// TwinCAT 3 PLC project PLC_LMP_VAC_current
// Title: LAMP PLC
// Author: A. Wallace, J. Yin and S. Stubbs
// Description: This version includes a longer needle valve purge time. Updated purge logic to quit the purge incase the interlocks on either VCN 40 VGP 40 or VIC 80 fail.
// ProgramVersion: 3.1.4020.1
// libraries:
//   LCLSVacuumLib,newest,SLAC
//   LCLSVacuumSerialDriverLib,newest,SLAC
//   Tc2_Standard,3.3.1.0,Beckhoff Automation GmbH
//   Tc2_SUPS,newest,Beckhoff Automation GmbH
//   Tc2_System,3.3.10.0,Beckhoff Automation GmbH
//   Tc2_Utilities,3.3.11.0,Beckhoff Automation GmbH
//   Tc3_Interfaces,3.3.0.0,Beckhoff Automation GmbH
//   Standard, * (System)
//   Tc2_SerialCom, * (Beckhoff Automation GmbH)
//   Tc3_Module, * (Beckhoff Automation GmbH)
// project tree:
//   Global Variables/ GVL.TcGVL, GVL_Autosave.TcGVL, GVL_COM_Buffers.TcGVL, GVL_Devices.TcGVL, GVL_IO.TcGVL, GVL_SerialIO.TcGVL
//   POUs/ Ext_Interlocks.TcPOU, MAIN.TcPOU, p_Initialize.TcPOU, p_SoftIOMap.TcPOU, p_ModbusMapRx.TcPOU, p_ModbusMapTx.TcPOU, p_GaugeSup.TcPOU, p_PTMSup.TcPOU, p_ValveSup.TcPOU, Encoders.TcPOU, p_Autosave.TcPOU, P_Serial_Com.TcPOU, P_Serial_PTM_IO.TcPOU
//   POUs/Functions/ FB_VRC_LAMP.TcPOU
//   / Standard.TcTTO, SerialIO.TcTTO
// real-time tasks:
//   TASK Standard: cycle T#10ms, priority 8, ADS port 351
//   TASK SerialIO: cycle T#5ms, priority 6, ADS port 352
// I/O:
//   DEVICE LAMP Fieldbus (EtherCAT), AmsNetId 5.21.50.18.2.1
//     Term 1 (EK1200) [EK1200-5000 EtherCAT Power supply (2A E-Bus)]
//       Term 2 (EL3064) [EL3064 4Ch. Ana. Input 0-10V]
//       Term 3 (EL3064) [EL3064 4Ch. Ana. Input 0-10V]
//       Term 4 (EL1008) [EL1008 8Ch. Dig. Input 24V, 3ms]
//       Term 5 (EL2008) [EL2008 8Ch. Dig. Output 24V, 0.5A]
//       Term 6 (EL2798) [EL2798 8Ch. Dig. Output 24V AC/DC, 2A, potential-free]
//       Term 7 (EL6731) [EL6731 PROFIBUS DP Master] (disabled)
//       Term 8 (EK1110) [EK1110 EtherCAT extension]
//     R10_A (EP6002-0002) [EP6002-0002 Interface (RS232/422/485)]
//     R10_B (EP6002-0002) [EP6002-0002 Interface (RS232/422/485)]
//     IC1-EB1 (EP6002-0002) [EP6002-0002 Interface (RS232/422/485)]
//     IC1-EB2 (EP3174-0002) [EP3174-0002 4Ch. Ana. Input +/-10V, 0-10V, 0/4-20mA configurable]
//     IC1-EB3 (EP2624-0002) [EP2624-0002 4Ch. Relay Output, NO (125V AC / 30V DC)]
//     IC1-EB4 (EP2339-0021) [EP2339-0021 16 Ch. Dig. Input/Output 24V, 0,5A, M8]
//     DET-EB1 (EP6002-0002) [EP6002-0002 Interface (RS232/422/485)]
//     DET-EB2 (EP3174-0002) [EP3174-0002 4Ch. Ana. Input +/-10V, 0-10V, 0/4-20mA configurable]
//     DET-EB3 (EP2624-0002) [EP2624-0002 4Ch. Relay Output, NO (125V AC / 30V DC)]
//     DET-EB4 (EP2339-0021) [EP2339-0021 16 Ch. Dig. Input/Output 24V, 0,5A, M8]
//     DET-EB5 (EP2624-0002) [EP2624-0002 4Ch. Relay Output, NO (125V AC / 30V DC)]
//     GJ1-EB1 (EP2624-0002) [EP2624-0002 4Ch. Relay Output, NO (125V AC / 30V DC)]
//     GJ-EB2 (EP3174-0002) [EP3174-0002 4Ch. Ana. Input +/-10V, 0-10V, 0/4-20mA configurable]
//     GJ-EB3 (EP2339-0021) [EP2339-0021 16 Ch. Dig. Input/Output 24V, 0,5A, M8]
//     GJ-EB4 (EP3174-0002) [EP3174-0002 4Ch. Ana. Input +/-10V, 0-10V, 0/4-20mA, +/-10mA configurable]
//     LRS-EB1 (EP3174-0002) [EP3174-0002 4Ch. Ana. Input +/-10V, 0-10V, 0/4-20mA configurable]
//     LRS-EB2 (EP3174-0002) [EP3174-0002 4Ch. Ana. Input +/-10V, 0-10V, 0/4-20mA, +/-10mA configurable]
//     LRS-EB3 (EP2339-0021) [EP2339-0021 16 Ch. Dig. Input/Output 24V, 0,5A, M8]
//     LRS-EB4 (EP2339-0021) [EP2339-0021 16 Ch. Dig. Input/Output 24V, 0,5A, M8]
//     H2E-EB1 (EP2339-0021) [EP2339-0021 16 Ch. Dig. Input/Output 24V, 0,5A, M8] (disabled)
//     H2E-EB2 (EP3174-0002) [EP3174-0002 4Ch. Ana. Input +/-10V, 0-10V, 0/4-20mA, +/-10mA configurable] (disabled)
//   DEVICE LAMP(EtherCAT Slave), AmsNetId 5.21.50.18.4.255
//   DEVICE Device 2 (EL6731) (disabled), AmsNetId 5.21.50.18.3.1
// variable links:
//   PLC_LMP_VAC_current/PLC_LMP_VAC_current Instance <-> LAMP Fieldbus (EtherCAT)/DET-EB1 (EP6002-0002)
//     SerialIO Inputs/GVL_SerialIO.DET_P1_stComIn/D[0] <-> COM TxPDO-Map Inputs Channel 1/Data In 0
//     SerialIO Inputs/GVL_SerialIO.DET_P1_stComIn/D[10] <-> COM TxPDO-Map Inputs Channel 1/Data In 10
//     SerialIO Inputs/GVL_SerialIO.DET_P1_stComIn/D[11] <-> COM TxPDO-Map Inputs Channel 1/Data In 11
//     SerialIO Inputs/GVL_SerialIO.DET_P1_stComIn/D[12] <-> COM TxPDO-Map Inputs Channel 1/Data In 12
//     SerialIO Inputs/GVL_SerialIO.DET_P1_stComIn/D[13] <-> COM TxPDO-Map Inputs Channel 1/Data In 13
//     SerialIO Inputs/GVL_SerialIO.DET_P1_stComIn/D[14] <-> COM TxPDO-Map Inputs Channel 1/Data In 14
//     SerialIO Inputs/GVL_SerialIO.DET_P1_stComIn/D[15] <-> COM TxPDO-Map Inputs Channel 1/Data In 15
//     SerialIO Inputs/GVL_SerialIO.DET_P1_stComIn/D[16] <-> COM TxPDO-Map Inputs Channel 1/Data In 16
//     SerialIO Inputs/GVL_SerialIO.DET_P1_stComIn/D[17] <-> COM TxPDO-Map Inputs Channel 1/Data In 17
//     SerialIO Inputs/GVL_SerialIO.DET_P1_stComIn/D[18] <-> COM TxPDO-Map Inputs Channel 1/Data In 18
//     SerialIO Inputs/GVL_SerialIO.DET_P1_stComIn/D[19] <-> COM TxPDO-Map Inputs Channel 1/Data In 19
//     SerialIO Inputs/GVL_SerialIO.DET_P1_stComIn/D[1] <-> COM TxPDO-Map Inputs Channel 1/Data In 1
//     SerialIO Inputs/GVL_SerialIO.DET_P1_stComIn/D[20] <-> COM TxPDO-Map Inputs Channel 1/Data In 20
//     SerialIO Inputs/GVL_SerialIO.DET_P1_stComIn/D[21] <-> COM TxPDO-Map Inputs Channel 1/Data In 21
//     SerialIO Inputs/GVL_SerialIO.DET_P1_stComIn/D[2] <-> COM TxPDO-Map Inputs Channel 1/Data In 2
//     SerialIO Inputs/GVL_SerialIO.DET_P1_stComIn/D[3] <-> COM TxPDO-Map Inputs Channel 1/Data In 3
//     SerialIO Inputs/GVL_SerialIO.DET_P1_stComIn/D[4] <-> COM TxPDO-Map Inputs Channel 1/Data In 4
//     SerialIO Inputs/GVL_SerialIO.DET_P1_stComIn/D[5] <-> COM TxPDO-Map Inputs Channel 1/Data In 5
//     SerialIO Inputs/GVL_SerialIO.DET_P1_stComIn/D[6] <-> COM TxPDO-Map Inputs Channel 1/Data In 6
//     SerialIO Inputs/GVL_SerialIO.DET_P1_stComIn/D[7] <-> COM TxPDO-Map Inputs Channel 1/Data In 7
//     SerialIO Inputs/GVL_SerialIO.DET_P1_stComIn/D[8] <-> COM TxPDO-Map Inputs Channel 1/Data In 8
//     SerialIO Inputs/GVL_SerialIO.DET_P1_stComIn/D[9] <-> COM TxPDO-Map Inputs Channel 1/Data In 9
//     SerialIO Inputs/GVL_SerialIO.DET_P2_stComIn/D[0] <-> COM TxPDO-Map Inputs Channel 2/Data In 0
//     SerialIO Inputs/GVL_SerialIO.DET_P2_stComIn/D[10] <-> COM TxPDO-Map Inputs Channel 2/Data In 10
//     SerialIO Inputs/GVL_SerialIO.DET_P2_stComIn/D[11] <-> COM TxPDO-Map Inputs Channel 2/Data In 11
//     SerialIO Inputs/GVL_SerialIO.DET_P2_stComIn/D[12] <-> COM TxPDO-Map Inputs Channel 2/Data In 12
//     SerialIO Inputs/GVL_SerialIO.DET_P2_stComIn/D[13] <-> COM TxPDO-Map Inputs Channel 2/Data In 13
//     SerialIO Inputs/GVL_SerialIO.DET_P2_stComIn/D[14] <-> COM TxPDO-Map Inputs Channel 2/Data In 14
//     SerialIO Inputs/GVL_SerialIO.DET_P2_stComIn/D[15] <-> COM TxPDO-Map Inputs Channel 2/Data In 15
//     SerialIO Inputs/GVL_SerialIO.DET_P2_stComIn/D[16] <-> COM TxPDO-Map Inputs Channel 2/Data In 16
//     SerialIO Inputs/GVL_SerialIO.DET_P2_stComIn/D[17] <-> COM TxPDO-Map Inputs Channel 2/Data In 17
//     SerialIO Inputs/GVL_SerialIO.DET_P2_stComIn/D[18] <-> COM TxPDO-Map Inputs Channel 2/Data In 18
//     SerialIO Inputs/GVL_SerialIO.DET_P2_stComIn/D[19] <-> COM TxPDO-Map Inputs Channel 2/Data In 19
//     SerialIO Inputs/GVL_SerialIO.DET_P2_stComIn/D[1] <-> COM TxPDO-Map Inputs Channel 2/Data In 1
//     SerialIO Inputs/GVL_SerialIO.DET_P2_stComIn/D[20] <-> COM TxPDO-Map Inputs Channel 2/Data In 20
//     SerialIO Inputs/GVL_SerialIO.DET_P2_stComIn/D[21] <-> COM TxPDO-Map Inputs Channel 2/Data In 21
//     SerialIO Inputs/GVL_SerialIO.DET_P2_stComIn/D[2] <-> COM TxPDO-Map Inputs Channel 2/Data In 2
//     SerialIO Inputs/GVL_SerialIO.DET_P2_stComIn/D[3] <-> COM TxPDO-Map Inputs Channel 2/Data In 3
//     SerialIO Inputs/GVL_SerialIO.DET_P2_stComIn/D[4] <-> COM TxPDO-Map Inputs Channel 2/Data In 4
//     SerialIO Inputs/GVL_SerialIO.DET_P2_stComIn/D[5] <-> COM TxPDO-Map Inputs Channel 2/Data In 5
//     SerialIO Inputs/GVL_SerialIO.DET_P2_stComIn/D[6] <-> COM TxPDO-Map Inputs Channel 2/Data In 6
//     SerialIO Inputs/GVL_SerialIO.DET_P2_stComIn/D[7] <-> COM TxPDO-Map Inputs Channel 2/Data In 7
//     SerialIO Inputs/GVL_SerialIO.DET_P2_stComIn/D[8] <-> COM TxPDO-Map Inputs Channel 2/Data In 8
//     SerialIO Inputs/GVL_SerialIO.DET_P2_stComIn/D[9] <-> COM TxPDO-Map Inputs Channel 2/Data In 9
//     SerialIO Inputs/GVL_SerialIO.DET_P1_stComIn/Status <-> COM TxPDO-Map Inputs Channel 1/Status
//     SerialIO Inputs/GVL_SerialIO.DET_P2_stComIn/Status <-> COM TxPDO-Map Inputs Channel 2/Status
//     SerialIO Outputs/GVL_SerialIO.DET_P1_stComOut/Ctrl <-> COM RxPDO-Map Outputs Channel 1/Ctrl
//     SerialIO Outputs/GVL_SerialIO.DET_P2_stComOut/Ctrl <-> COM RxPDO-Map Outputs Channel 2/Ctrl
//     SerialIO Outputs/GVL_SerialIO.DET_P1_stComOut/D[0] <-> COM RxPDO-Map Outputs Channel 1/Data Out 0
//     SerialIO Outputs/GVL_SerialIO.DET_P1_stComOut/D[10] <-> COM RxPDO-Map Outputs Channel 1/Data Out 10
//     SerialIO Outputs/GVL_SerialIO.DET_P1_stComOut/D[11] <-> COM RxPDO-Map Outputs Channel 1/Data Out 11
//     SerialIO Outputs/GVL_SerialIO.DET_P1_stComOut/D[12] <-> COM RxPDO-Map Outputs Channel 1/Data Out 12
//     SerialIO Outputs/GVL_SerialIO.DET_P1_stComOut/D[13] <-> COM RxPDO-Map Outputs Channel 1/Data Out 13
//     SerialIO Outputs/GVL_SerialIO.DET_P1_stComOut/D[14] <-> COM RxPDO-Map Outputs Channel 1/Data Out 14
//     SerialIO Outputs/GVL_SerialIO.DET_P1_stComOut/D[15] <-> COM RxPDO-Map Outputs Channel 1/Data Out 15
//     SerialIO Outputs/GVL_SerialIO.DET_P1_stComOut/D[16] <-> COM RxPDO-Map Outputs Channel 1/Data Out 16
//     SerialIO Outputs/GVL_SerialIO.DET_P1_stComOut/D[17] <-> COM RxPDO-Map Outputs Channel 1/Data Out 17
//     SerialIO Outputs/GVL_SerialIO.DET_P1_stComOut/D[18] <-> COM RxPDO-Map Outputs Channel 1/Data Out 18
//     SerialIO Outputs/GVL_SerialIO.DET_P1_stComOut/D[19] <-> COM RxPDO-Map Outputs Channel 1/Data Out 19
//     SerialIO Outputs/GVL_SerialIO.DET_P1_stComOut/D[1] <-> COM RxPDO-Map Outputs Channel 1/Data Out 1
//     SerialIO Outputs/GVL_SerialIO.DET_P1_stComOut/D[20] <-> COM RxPDO-Map Outputs Channel 1/Data Out 20
//     SerialIO Outputs/GVL_SerialIO.DET_P1_stComOut/D[21] <-> COM RxPDO-Map Outputs Channel 1/Data Out 21
//     SerialIO Outputs/GVL_SerialIO.DET_P1_stComOut/D[2] <-> COM RxPDO-Map Outputs Channel 1/Data Out 2
//     SerialIO Outputs/GVL_SerialIO.DET_P1_stComOut/D[3] <-> COM RxPDO-Map Outputs Channel 1/Data Out 3
//     SerialIO Outputs/GVL_SerialIO.DET_P1_stComOut/D[4] <-> COM RxPDO-Map Outputs Channel 1/Data Out 4
//     SerialIO Outputs/GVL_SerialIO.DET_P1_stComOut/D[5] <-> COM RxPDO-Map Outputs Channel 1/Data Out 5
//     SerialIO Outputs/GVL_SerialIO.DET_P1_stComOut/D[6] <-> COM RxPDO-Map Outputs Channel 1/Data Out 6
//     SerialIO Outputs/GVL_SerialIO.DET_P1_stComOut/D[7] <-> COM RxPDO-Map Outputs Channel 1/Data Out 7
//     SerialIO Outputs/GVL_SerialIO.DET_P1_stComOut/D[8] <-> COM RxPDO-Map Outputs Channel 1/Data Out 8
//     SerialIO Outputs/GVL_SerialIO.DET_P1_stComOut/D[9] <-> COM RxPDO-Map Outputs Channel 1/Data Out 9
//     SerialIO Outputs/GVL_SerialIO.DET_P2_stComOut/D[0] <-> COM RxPDO-Map Outputs Channel 2/Data Out 0
//     SerialIO Outputs/GVL_SerialIO.DET_P2_stComOut/D[10] <-> COM RxPDO-Map Outputs Channel 2/Data Out 10
//     SerialIO Outputs/GVL_SerialIO.DET_P2_stComOut/D[11] <-> COM RxPDO-Map Outputs Channel 2/Data Out 11
//     SerialIO Outputs/GVL_SerialIO.DET_P2_stComOut/D[12] <-> COM RxPDO-Map Outputs Channel 2/Data Out 12
//     SerialIO Outputs/GVL_SerialIO.DET_P2_stComOut/D[13] <-> COM RxPDO-Map Outputs Channel 2/Data Out 13
//     SerialIO Outputs/GVL_SerialIO.DET_P2_stComOut/D[14] <-> COM RxPDO-Map Outputs Channel 2/Data Out 14
//     SerialIO Outputs/GVL_SerialIO.DET_P2_stComOut/D[15] <-> COM RxPDO-Map Outputs Channel 2/Data Out 15
//     SerialIO Outputs/GVL_SerialIO.DET_P2_stComOut/D[16] <-> COM RxPDO-Map Outputs Channel 2/Data Out 16
//     SerialIO Outputs/GVL_SerialIO.DET_P2_stComOut/D[17] <-> COM RxPDO-Map Outputs Channel 2/Data Out 17
//     SerialIO Outputs/GVL_SerialIO.DET_P2_stComOut/D[18] <-> COM RxPDO-Map Outputs Channel 2/Data Out 18
//     SerialIO Outputs/GVL_SerialIO.DET_P2_stComOut/D[19] <-> COM RxPDO-Map Outputs Channel 2/Data Out 19
//     SerialIO Outputs/GVL_SerialIO.DET_P2_stComOut/D[1] <-> COM RxPDO-Map Outputs Channel 2/Data Out 1
//     SerialIO Outputs/GVL_SerialIO.DET_P2_stComOut/D[20] <-> COM RxPDO-Map Outputs Channel 2/Data Out 20
//     SerialIO Outputs/GVL_SerialIO.DET_P2_stComOut/D[21] <-> COM RxPDO-Map Outputs Channel 2/Data Out 21
//     SerialIO Outputs/GVL_SerialIO.DET_P2_stComOut/D[2] <-> COM RxPDO-Map Outputs Channel 2/Data Out 2
//     SerialIO Outputs/GVL_SerialIO.DET_P2_stComOut/D[3] <-> COM RxPDO-Map Outputs Channel 2/Data Out 3
//     SerialIO Outputs/GVL_SerialIO.DET_P2_stComOut/D[4] <-> COM RxPDO-Map Outputs Channel 2/Data Out 4
//     SerialIO Outputs/GVL_SerialIO.DET_P2_stComOut/D[5] <-> COM RxPDO-Map Outputs Channel 2/Data Out 5
//     SerialIO Outputs/GVL_SerialIO.DET_P2_stComOut/D[6] <-> COM RxPDO-Map Outputs Channel 2/Data Out 6
//     SerialIO Outputs/GVL_SerialIO.DET_P2_stComOut/D[7] <-> COM RxPDO-Map Outputs Channel 2/Data Out 7
//     SerialIO Outputs/GVL_SerialIO.DET_P2_stComOut/D[8] <-> COM RxPDO-Map Outputs Channel 2/Data Out 8
//     SerialIO Outputs/GVL_SerialIO.DET_P2_stComOut/D[9] <-> COM RxPDO-Map Outputs Channel 2/Data Out 9
//   PLC_LMP_VAC_current/PLC_LMP_VAC_current Instance <-> LAMP Fieldbus (EtherCAT)/DET-EB2 (EP3174-0002)
//     Standard Inputs/GVL_IO.AI_DET_EB2Ch01 <-> AI Standard Channel 1/Value
//     Standard Inputs/GVL_IO.AI_DET_EB2Ch02 <-> AI Standard Channel 2/Value
//     Standard Inputs/GVL_IO.AI_DET_EB2Ch03 <-> AI Standard Channel 3/Value
//     Standard Inputs/GVL_IO.AI_DET_EB2Ch04 <-> AI Standard Channel 4/Value
//   PLC_LMP_VAC_current/PLC_LMP_VAC_current Instance <-> LAMP Fieldbus (EtherCAT)/DET-EB3 (EP2624-0002)
//     Standard Outputs/GVL_IO.RelayO_DET_EB3Ch01 <-> Channel 1/Output
//     Standard Outputs/GVL_IO.RelayO_DET_EB3Ch02 <-> Channel 2/Output
//     Standard Outputs/GVL_IO.RelayO_DET_EB3Ch03 <-> Channel 3/Output
//     Standard Outputs/GVL_IO.RelayO_DET_EB3Ch04 <-> Channel 4/Output
//   PLC_LMP_VAC_current/PLC_LMP_VAC_current Instance <-> LAMP Fieldbus (EtherCAT)/DET-EB4 (EP2339-0021)
//     Standard Inputs/GVL_IO.DiscIO_DET_EB4Ch02 <-> Channel 2/Input
//     Standard Inputs/GVL_IO.DiscIO_DET_EB4Ch03 <-> Channel 3/Input
//     Standard Inputs/GVL_IO.DiscIO_DET_EB4Ch05 <-> Channel 5/Input
//     Standard Inputs/GVL_IO.DiscIO_DET_EB4Ch06 <-> Channel 6/Input
//     Standard Inputs/GVL_IO.DiscIO_DET_EB4Ch08 <-> Channel 8/Input
//     Standard Inputs/GVL_IO.DiscIO_DET_EB4Ch09 <-> Channel 9/Input
//     Standard Inputs/GVL_IO.DiscIO_DET_EB4Ch11 <-> Channel 11/Input
//     Standard Inputs/GVL_IO.DiscIO_DET_EB4Ch12 <-> Channel 12/Input
//     Standard Inputs/GVL_IO.DiscIO_DET_EB4Ch14 <-> Channel 14/Input
//     Standard Inputs/GVL_IO.DiscIO_DET_EB4Ch15 <-> Channel 15/Input
//     Standard Inputs/GVL_IO.DiscIO_DET_EB4Ch16 <-> Channel 16/Input
//     Standard Outputs/GVL_IO.DiscIO_DET_EB4Ch01 <-> Channel 17/Output
//     Standard Outputs/GVL_IO.DiscIO_DET_EB4Ch04 <-> Channel 20/Output
//     Standard Outputs/GVL_IO.DiscIO_DET_EB4Ch07 <-> Channel 23/Output
//     Standard Outputs/GVL_IO.DiscIO_DET_EB4Ch10 <-> Channel 26/Output
//     Standard Outputs/GVL_IO.DiscIO_DET_EB4Ch13 <-> Channel 29/Output
//   PLC_LMP_VAC_current/PLC_LMP_VAC_current Instance <-> LAMP Fieldbus (EtherCAT)/DET-EB5 (EP2624-0002)
//     Standard Outputs/GVL_IO.RelayO_DET_EB5Ch01 <-> Channel 1/Output
//     Standard Outputs/GVL_IO.RelayO_DET_EB5Ch02 <-> Channel 2/Output
//     Standard Outputs/GVL_IO.RelayO_DET_EB5Ch03 <-> Channel 3/Output
//     Standard Outputs/GVL_IO.RelayO_DET_EB5Ch04 <-> Channel 4/Output
//   PLC_LMP_VAC_current/PLC_LMP_VAC_current Instance <-> LAMP Fieldbus (EtherCAT)/GJ-EB2 (EP3174-0002)
//     Standard Inputs/GVL_IO.AI_GJ_EB2Ch01 <-> AI Standard Channel 1/Value
//     Standard Inputs/GVL_IO.AI_GJ_EB2Ch02 <-> AI Standard Channel 2/Value
//     Standard Inputs/GVL_IO.AI_GJ_EB2Ch03 <-> AI Standard Channel 3/Value
//     Standard Inputs/GVL_IO.AI_GJ_EB2Ch04 <-> AI Standard Channel 4/Value
//   PLC_LMP_VAC_current/PLC_LMP_VAC_current Instance <-> LAMP Fieldbus (EtherCAT)/GJ-EB3 (EP2339-0021)
//     Standard Inputs/GVL_IO.DiscIO_GJ_EB3Ch02 <-> Channel 2/Input
//     Standard Inputs/GVL_IO.DiscIO_GJ_EB3Ch03 <-> Channel 3/Input
//     Standard Inputs/GVL_IO.DiscIO_GJ_EB3Ch05 <-> Channel 5/Input
//     Standard Inputs/GVL_IO.DiscIO_GJ_EB3Ch06 <-> Channel 6/Input
//     Standard Inputs/GVL_IO.DiscIO_GJ_EB3Ch08 <-> Channel 8/Input
//     Standard Inputs/GVL_IO.DiscIO_GJ_EB3Ch09 <-> Channel 9/Input
//     Standard Inputs/GVL_IO.DiscIO_GJ_EB3Ch11 <-> Channel 11/Input
//     Standard Inputs/GVL_IO.DiscIO_GJ_EB3Ch12 <-> Channel 12/Input
//     Standard Inputs/GVL_IO.DiscIO_GJ_EB3Ch14 <-> Channel 14/Input
//     Standard Inputs/GVL_IO.DiscIO_GJ_EB3Ch15 <-> Channel 15/Input
//     Standard Inputs/GVL_IO.DiscIO_GJ_EB3Ch16 <-> Channel 16/Input
//     Standard Outputs/GVL_IO.DiscIO_GJ_EB3Ch01 <-> Channel 17/Output
//     Standard Outputs/GVL_IO.DiscIO_GJ_EB3Ch04 <-> Channel 20/Output
//     Standard Outputs/GVL_IO.DiscIO_GJ_EB3Ch07 <-> Channel 23/Output
//     Standard Outputs/GVL_IO.DiscIO_GJ_EB3Ch10 <-> Channel 26/Output
//     Standard Outputs/GVL_IO.DiscIO_GJ_EB3Ch13 <-> Channel 29/Output
//   PLC_LMP_VAC_current/PLC_LMP_VAC_current Instance <-> LAMP Fieldbus (EtherCAT)/GJ-EB4 (EP3174-0002)
//     Standard Inputs/GVL_IO.AI_GJ_EB4Ch01 <-> AI Standard Channel 1/Value
//     Standard Inputs/GVL_IO.AI_GJ_EB4Ch02 <-> AI Standard Channel 2/Value
//     Standard Inputs/GVL_IO.AI_GJ_EB4Ch03 <-> AI Standard Channel 3/Value
//     Standard Inputs/GVL_IO.AI_GJ_EB4Ch04 <-> AI Standard Channel 4/Value
//   PLC_LMP_VAC_current/PLC_LMP_VAC_current Instance <-> LAMP Fieldbus (EtherCAT)/GJ1-EB1 (EP2624-0002)
//     Standard Outputs/GVL_IO.RelayO_GJ_EB1Ch01 <-> Channel 1/Output
//     Standard Outputs/GVL_IO.RelayO_GJ_EB1Ch02 <-> Channel 2/Output
//     Standard Outputs/GVL_IO.RelayO_GJ_EB1Ch03 <-> Channel 3/Output
//     Standard Outputs/GVL_IO.RelayO_GJ_EB1Ch04 <-> Channel 4/Output
//   PLC_LMP_VAC_current/PLC_LMP_VAC_current Instance <-> LAMP Fieldbus (EtherCAT)/H2E-EB1 (EP2339-0021)
//     Standard Inputs/GVL_IO.DiscIO_H2E_EB1Ch02 <-> Channel 2/Input
//     Standard Inputs/GVL_IO.DiscIO_H2E_EB1Ch03 <-> Channel 3/Input
//     Standard Inputs/GVL_IO.DiscIO_H2E_EB1Ch05 <-> Channel 5/Input
//     Standard Inputs/GVL_IO.DiscIO_H2E_EB1Ch06 <-> Channel 6/Input
//     Standard Inputs/GVL_IO.DiscIO_H2E_EB1Ch08 <-> Channel 8/Input
//     Standard Inputs/GVL_IO.DiscIO_H2E_EB1Ch09 <-> Channel 9/Input
//     Standard Inputs/GVL_IO.DiscIO_H2E_EB1Ch11 <-> Channel 11/Input
//     Standard Inputs/GVL_IO.DiscIO_H2E_EB1Ch12 <-> Channel 12/Input
//     Standard Inputs/GVL_IO.DiscIO_H2E_EB1Ch14 <-> Channel 14/Input
//     Standard Inputs/GVL_IO.DiscIO_H2E_EB1Ch15 <-> Channel 15/Input
//     Standard Inputs/GVL_IO.DiscIO_H2E_EB1Ch16 <-> Channel 16/Input
//     Standard Outputs/GVL_IO.DiscIO_H2E_EB1Ch01 <-> Channel 17/Output
//     Standard Outputs/GVL_IO.DiscIO_H2E_EB1Ch04 <-> Channel 20/Output
//     Standard Outputs/GVL_IO.DiscIO_H2E_EB1Ch07 <-> Channel 23/Output
//     Standard Outputs/GVL_IO.DiscIO_H2E_EB1Ch10 <-> Channel 26/Output
//     Standard Outputs/GVL_IO.DiscIO_H2E_EB1Ch13 <-> Channel 29/Output
//   PLC_LMP_VAC_current/PLC_LMP_VAC_current Instance <-> LAMP Fieldbus (EtherCAT)/H2E-EB2 (EP3174-0002)
//     Standard Inputs/GVL_IO.AI_H2E_EB2Ch01 <-> AI Standard Channel 1/Value
//     Standard Inputs/GVL_IO.AI_H2E_EB2Ch02 <-> AI Standard Channel 2/Value
//     Standard Inputs/GVL_IO.AI_H2E_EB2Ch03 <-> AI Standard Channel 3/Value
//     Standard Inputs/GVL_IO.AI_H2E_EB2Ch04 <-> AI Standard Channel 4/Value
//   PLC_LMP_VAC_current/PLC_LMP_VAC_current Instance <-> LAMP Fieldbus (EtherCAT)/IC1-EB1 (EP6002-0002)
//     SerialIO Inputs/GVL_SerialIO.IC_P1_stComIn/D[0] <-> COM TxPDO-Map Inputs Channel 1/Data In 0
//     SerialIO Inputs/GVL_SerialIO.IC_P1_stComIn/D[10] <-> COM TxPDO-Map Inputs Channel 1/Data In 10
//     SerialIO Inputs/GVL_SerialIO.IC_P1_stComIn/D[11] <-> COM TxPDO-Map Inputs Channel 1/Data In 11
//     SerialIO Inputs/GVL_SerialIO.IC_P1_stComIn/D[12] <-> COM TxPDO-Map Inputs Channel 1/Data In 12
//     SerialIO Inputs/GVL_SerialIO.IC_P1_stComIn/D[13] <-> COM TxPDO-Map Inputs Channel 1/Data In 13
//     SerialIO Inputs/GVL_SerialIO.IC_P1_stComIn/D[14] <-> COM TxPDO-Map Inputs Channel 1/Data In 14
//     SerialIO Inputs/GVL_SerialIO.IC_P1_stComIn/D[15] <-> COM TxPDO-Map Inputs Channel 1/Data In 15
//     SerialIO Inputs/GVL_SerialIO.IC_P1_stComIn/D[16] <-> COM TxPDO-Map Inputs Channel 1/Data In 16
//     SerialIO Inputs/GVL_SerialIO.IC_P1_stComIn/D[17] <-> COM TxPDO-Map Inputs Channel 1/Data In 17
//     SerialIO Inputs/GVL_SerialIO.IC_P1_stComIn/D[18] <-> COM TxPDO-Map Inputs Channel 1/Data In 18
//     SerialIO Inputs/GVL_SerialIO.IC_P1_stComIn/D[19] <-> COM TxPDO-Map Inputs Channel 1/Data In 19
//     SerialIO Inputs/GVL_SerialIO.IC_P1_stComIn/D[1] <-> COM TxPDO-Map Inputs Channel 1/Data In 1
//     SerialIO Inputs/GVL_SerialIO.IC_P1_stComIn/D[20] <-> COM TxPDO-Map Inputs Channel 1/Data In 20
//     SerialIO Inputs/GVL_SerialIO.IC_P1_stComIn/D[21] <-> COM TxPDO-Map Inputs Channel 1/Data In 21
//     SerialIO Inputs/GVL_SerialIO.IC_P1_stComIn/D[2] <-> COM TxPDO-Map Inputs Channel 1/Data In 2
//     SerialIO Inputs/GVL_SerialIO.IC_P1_stComIn/D[3] <-> COM TxPDO-Map Inputs Channel 1/Data In 3
//     SerialIO Inputs/GVL_SerialIO.IC_P1_stComIn/D[4] <-> COM TxPDO-Map Inputs Channel 1/Data In 4
//     SerialIO Inputs/GVL_SerialIO.IC_P1_stComIn/D[5] <-> COM TxPDO-Map Inputs Channel 1/Data In 5
//     SerialIO Inputs/GVL_SerialIO.IC_P1_stComIn/D[6] <-> COM TxPDO-Map Inputs Channel 1/Data In 6
//     SerialIO Inputs/GVL_SerialIO.IC_P1_stComIn/D[7] <-> COM TxPDO-Map Inputs Channel 1/Data In 7
//     SerialIO Inputs/GVL_SerialIO.IC_P1_stComIn/D[8] <-> COM TxPDO-Map Inputs Channel 1/Data In 8
//     SerialIO Inputs/GVL_SerialIO.IC_P1_stComIn/D[9] <-> COM TxPDO-Map Inputs Channel 1/Data In 9
//     SerialIO Inputs/GVL_SerialIO.IC_P2_stComIn/D[0] <-> COM TxPDO-Map Inputs Channel 2/Data In 0
//     SerialIO Inputs/GVL_SerialIO.IC_P2_stComIn/D[10] <-> COM TxPDO-Map Inputs Channel 2/Data In 10
//     SerialIO Inputs/GVL_SerialIO.IC_P2_stComIn/D[11] <-> COM TxPDO-Map Inputs Channel 2/Data In 11
//     SerialIO Inputs/GVL_SerialIO.IC_P2_stComIn/D[12] <-> COM TxPDO-Map Inputs Channel 2/Data In 12
//     SerialIO Inputs/GVL_SerialIO.IC_P2_stComIn/D[13] <-> COM TxPDO-Map Inputs Channel 2/Data In 13
//     SerialIO Inputs/GVL_SerialIO.IC_P2_stComIn/D[14] <-> COM TxPDO-Map Inputs Channel 2/Data In 14
//     SerialIO Inputs/GVL_SerialIO.IC_P2_stComIn/D[15] <-> COM TxPDO-Map Inputs Channel 2/Data In 15
//     SerialIO Inputs/GVL_SerialIO.IC_P2_stComIn/D[16] <-> COM TxPDO-Map Inputs Channel 2/Data In 16
//     SerialIO Inputs/GVL_SerialIO.IC_P2_stComIn/D[17] <-> COM TxPDO-Map Inputs Channel 2/Data In 17
//     SerialIO Inputs/GVL_SerialIO.IC_P2_stComIn/D[18] <-> COM TxPDO-Map Inputs Channel 2/Data In 18
//     SerialIO Inputs/GVL_SerialIO.IC_P2_stComIn/D[19] <-> COM TxPDO-Map Inputs Channel 2/Data In 19
//     SerialIO Inputs/GVL_SerialIO.IC_P2_stComIn/D[1] <-> COM TxPDO-Map Inputs Channel 2/Data In 1
//     SerialIO Inputs/GVL_SerialIO.IC_P2_stComIn/D[20] <-> COM TxPDO-Map Inputs Channel 2/Data In 20
//     SerialIO Inputs/GVL_SerialIO.IC_P2_stComIn/D[21] <-> COM TxPDO-Map Inputs Channel 2/Data In 21
//     SerialIO Inputs/GVL_SerialIO.IC_P2_stComIn/D[2] <-> COM TxPDO-Map Inputs Channel 2/Data In 2
//     SerialIO Inputs/GVL_SerialIO.IC_P2_stComIn/D[3] <-> COM TxPDO-Map Inputs Channel 2/Data In 3
//     SerialIO Inputs/GVL_SerialIO.IC_P2_stComIn/D[4] <-> COM TxPDO-Map Inputs Channel 2/Data In 4
//     SerialIO Inputs/GVL_SerialIO.IC_P2_stComIn/D[5] <-> COM TxPDO-Map Inputs Channel 2/Data In 5
//     SerialIO Inputs/GVL_SerialIO.IC_P2_stComIn/D[6] <-> COM TxPDO-Map Inputs Channel 2/Data In 6
//     SerialIO Inputs/GVL_SerialIO.IC_P2_stComIn/D[7] <-> COM TxPDO-Map Inputs Channel 2/Data In 7
//     SerialIO Inputs/GVL_SerialIO.IC_P2_stComIn/D[8] <-> COM TxPDO-Map Inputs Channel 2/Data In 8
//     SerialIO Inputs/GVL_SerialIO.IC_P2_stComIn/D[9] <-> COM TxPDO-Map Inputs Channel 2/Data In 9
//     SerialIO Inputs/GVL_SerialIO.IC_P1_stComIn/Status <-> COM TxPDO-Map Inputs Channel 1/Status
//     SerialIO Inputs/GVL_SerialIO.IC_P2_stComIn/Status <-> COM TxPDO-Map Inputs Channel 2/Status
//     SerialIO Outputs/GVL_SerialIO.IC_P1_stComOut/Ctrl <-> COM RxPDO-Map Outputs Channel 1/Ctrl
//     SerialIO Outputs/GVL_SerialIO.IC_P2_stComOut/Ctrl <-> COM RxPDO-Map Outputs Channel 2/Ctrl
//     SerialIO Outputs/GVL_SerialIO.IC_P1_stComOut/D[0] <-> COM RxPDO-Map Outputs Channel 1/Data Out 0
//     SerialIO Outputs/GVL_SerialIO.IC_P1_stComOut/D[10] <-> COM RxPDO-Map Outputs Channel 1/Data Out 10
//     SerialIO Outputs/GVL_SerialIO.IC_P1_stComOut/D[11] <-> COM RxPDO-Map Outputs Channel 1/Data Out 11
//     SerialIO Outputs/GVL_SerialIO.IC_P1_stComOut/D[12] <-> COM RxPDO-Map Outputs Channel 1/Data Out 12
//     SerialIO Outputs/GVL_SerialIO.IC_P1_stComOut/D[13] <-> COM RxPDO-Map Outputs Channel 1/Data Out 13
//     SerialIO Outputs/GVL_SerialIO.IC_P1_stComOut/D[14] <-> COM RxPDO-Map Outputs Channel 1/Data Out 14
//     SerialIO Outputs/GVL_SerialIO.IC_P1_stComOut/D[15] <-> COM RxPDO-Map Outputs Channel 1/Data Out 15
//     SerialIO Outputs/GVL_SerialIO.IC_P1_stComOut/D[16] <-> COM RxPDO-Map Outputs Channel 1/Data Out 16
//     SerialIO Outputs/GVL_SerialIO.IC_P1_stComOut/D[17] <-> COM RxPDO-Map Outputs Channel 1/Data Out 17
//     SerialIO Outputs/GVL_SerialIO.IC_P1_stComOut/D[18] <-> COM RxPDO-Map Outputs Channel 1/Data Out 18
//     SerialIO Outputs/GVL_SerialIO.IC_P1_stComOut/D[19] <-> COM RxPDO-Map Outputs Channel 1/Data Out 19
//     SerialIO Outputs/GVL_SerialIO.IC_P1_stComOut/D[1] <-> COM RxPDO-Map Outputs Channel 1/Data Out 1
//     SerialIO Outputs/GVL_SerialIO.IC_P1_stComOut/D[20] <-> COM RxPDO-Map Outputs Channel 1/Data Out 20
//     SerialIO Outputs/GVL_SerialIO.IC_P1_stComOut/D[21] <-> COM RxPDO-Map Outputs Channel 1/Data Out 21
//     SerialIO Outputs/GVL_SerialIO.IC_P1_stComOut/D[2] <-> COM RxPDO-Map Outputs Channel 1/Data Out 2
//     SerialIO Outputs/GVL_SerialIO.IC_P1_stComOut/D[3] <-> COM RxPDO-Map Outputs Channel 1/Data Out 3
//     SerialIO Outputs/GVL_SerialIO.IC_P1_stComOut/D[4] <-> COM RxPDO-Map Outputs Channel 1/Data Out 4
//     SerialIO Outputs/GVL_SerialIO.IC_P1_stComOut/D[5] <-> COM RxPDO-Map Outputs Channel 1/Data Out 5
//     SerialIO Outputs/GVL_SerialIO.IC_P1_stComOut/D[6] <-> COM RxPDO-Map Outputs Channel 1/Data Out 6
//     SerialIO Outputs/GVL_SerialIO.IC_P1_stComOut/D[7] <-> COM RxPDO-Map Outputs Channel 1/Data Out 7
//     SerialIO Outputs/GVL_SerialIO.IC_P1_stComOut/D[8] <-> COM RxPDO-Map Outputs Channel 1/Data Out 8
//     SerialIO Outputs/GVL_SerialIO.IC_P1_stComOut/D[9] <-> COM RxPDO-Map Outputs Channel 1/Data Out 9
//     SerialIO Outputs/GVL_SerialIO.IC_P2_stComOut/D[0] <-> COM RxPDO-Map Outputs Channel 2/Data Out 0
//     SerialIO Outputs/GVL_SerialIO.IC_P2_stComOut/D[10] <-> COM RxPDO-Map Outputs Channel 2/Data Out 10
//     SerialIO Outputs/GVL_SerialIO.IC_P2_stComOut/D[11] <-> COM RxPDO-Map Outputs Channel 2/Data Out 11
//     SerialIO Outputs/GVL_SerialIO.IC_P2_stComOut/D[12] <-> COM RxPDO-Map Outputs Channel 2/Data Out 12
//     SerialIO Outputs/GVL_SerialIO.IC_P2_stComOut/D[13] <-> COM RxPDO-Map Outputs Channel 2/Data Out 13
//     SerialIO Outputs/GVL_SerialIO.IC_P2_stComOut/D[14] <-> COM RxPDO-Map Outputs Channel 2/Data Out 14
//     SerialIO Outputs/GVL_SerialIO.IC_P2_stComOut/D[15] <-> COM RxPDO-Map Outputs Channel 2/Data Out 15
//     SerialIO Outputs/GVL_SerialIO.IC_P2_stComOut/D[16] <-> COM RxPDO-Map Outputs Channel 2/Data Out 16
//     SerialIO Outputs/GVL_SerialIO.IC_P2_stComOut/D[17] <-> COM RxPDO-Map Outputs Channel 2/Data Out 17
//     SerialIO Outputs/GVL_SerialIO.IC_P2_stComOut/D[18] <-> COM RxPDO-Map Outputs Channel 2/Data Out 18
//     SerialIO Outputs/GVL_SerialIO.IC_P2_stComOut/D[19] <-> COM RxPDO-Map Outputs Channel 2/Data Out 19
//     SerialIO Outputs/GVL_SerialIO.IC_P2_stComOut/D[1] <-> COM RxPDO-Map Outputs Channel 2/Data Out 1
//     SerialIO Outputs/GVL_SerialIO.IC_P2_stComOut/D[20] <-> COM RxPDO-Map Outputs Channel 2/Data Out 20
//     SerialIO Outputs/GVL_SerialIO.IC_P2_stComOut/D[21] <-> COM RxPDO-Map Outputs Channel 2/Data Out 21
//     SerialIO Outputs/GVL_SerialIO.IC_P2_stComOut/D[2] <-> COM RxPDO-Map Outputs Channel 2/Data Out 2
//     SerialIO Outputs/GVL_SerialIO.IC_P2_stComOut/D[3] <-> COM RxPDO-Map Outputs Channel 2/Data Out 3
//     SerialIO Outputs/GVL_SerialIO.IC_P2_stComOut/D[4] <-> COM RxPDO-Map Outputs Channel 2/Data Out 4
//     SerialIO Outputs/GVL_SerialIO.IC_P2_stComOut/D[5] <-> COM RxPDO-Map Outputs Channel 2/Data Out 5
//     SerialIO Outputs/GVL_SerialIO.IC_P2_stComOut/D[6] <-> COM RxPDO-Map Outputs Channel 2/Data Out 6
//     SerialIO Outputs/GVL_SerialIO.IC_P2_stComOut/D[7] <-> COM RxPDO-Map Outputs Channel 2/Data Out 7
//     SerialIO Outputs/GVL_SerialIO.IC_P2_stComOut/D[8] <-> COM RxPDO-Map Outputs Channel 2/Data Out 8
//     SerialIO Outputs/GVL_SerialIO.IC_P2_stComOut/D[9] <-> COM RxPDO-Map Outputs Channel 2/Data Out 9
//   PLC_LMP_VAC_current/PLC_LMP_VAC_current Instance <-> LAMP Fieldbus (EtherCAT)/IC1-EB2 (EP3174-0002)
//     Standard Inputs/GVL_IO.AI_IC_EB2Ch01 <-> AI Standard Channel 1/Value
//     Standard Inputs/GVL_IO.AI_IC_EB2Ch02 <-> AI Standard Channel 2/Value
//     Standard Inputs/GVL_IO.AI_IC_EB2Ch03 <-> AI Standard Channel 3/Value
//     Standard Inputs/GVL_IO.AI_IC_EB2Ch04 <-> AI Standard Channel 4/Value
//   PLC_LMP_VAC_current/PLC_LMP_VAC_current Instance <-> LAMP Fieldbus (EtherCAT)/IC1-EB3 (EP2624-0002)
//     Standard Outputs/GVL_IO.RelayO_IC_EB3Ch01 <-> Channel 1/Output
//     Standard Outputs/GVL_IO.RelayO_IC_EB3Ch02 <-> Channel 2/Output
//     Standard Outputs/GVL_IO.RelayO_IC_EB3Ch03 <-> Channel 3/Output
//     Standard Outputs/GVL_IO.RelayO_IC_EB3Ch04 <-> Channel 4/Output
//   PLC_LMP_VAC_current/PLC_LMP_VAC_current Instance <-> LAMP Fieldbus (EtherCAT)/IC1-EB4 (EP2339-0021)
//     Standard Inputs/GVL_IO.DiscIO_IC_EB4Ch02 <-> Channel 2/Input
//     Standard Inputs/GVL_IO.DiscIO_IC_EB4Ch03 <-> Channel 3/Input
//     Standard Inputs/GVL_IO.DiscIO_IC_EB4Ch05 <-> Channel 5/Input
//     Standard Inputs/GVL_IO.DiscIO_IC_EB4Ch06 <-> Channel 6/Input
//     Standard Inputs/GVL_IO.DiscIO_IC_EB4Ch08 <-> Channel 8/Input
//     Standard Inputs/GVL_IO.DiscIO_IC_EB4Ch09 <-> Channel 9/Input
//     Standard Inputs/GVL_IO.DiscIO_IC_EB4Ch11 <-> Channel 11/Input
//     Standard Inputs/GVL_IO.DiscIO_IC_EB4Ch12 <-> Channel 12/Input
//     Standard Inputs/GVL_IO.DiscIO_IC_EB4Ch14 <-> Channel 14/Input
//     Standard Inputs/GVL_IO.DiscIO_IC_EB4Ch15 <-> Channel 15/Input
//     Standard Inputs/GVL_IO.DiscIO_IC_EB4Ch16 <-> Channel 16/Input
//     Standard Outputs/GVL_IO.DiscIO_IC_EB4Ch01 <-> Channel 17/Output
//     Standard Outputs/GVL_IO.DiscIO_IC_EB4Ch04 <-> Channel 20/Output
//     Standard Outputs/GVL_IO.DiscIO_IC_EB4Ch07 <-> Channel 23/Output
//     Standard Outputs/GVL_IO.DiscIO_IC_EB4Ch10 <-> Channel 26/Output
//     Standard Outputs/GVL_IO.DiscIO_IC_EB4Ch13 <-> Channel 29/Output
//   PLC_LMP_VAC_current/PLC_LMP_VAC_current Instance <-> LAMP Fieldbus (EtherCAT)/LRS-EB1 (EP3174-0002)
//     Standard Inputs/GVL_IO.AI_LRS_EB1Ch01 <-> AI Standard Channel 1/Value
//     Standard Inputs/GVL_IO.AI_LRS_EB1Ch02 <-> AI Standard Channel 2/Value
//     Standard Inputs/GVL_IO.AI_LRS_EB1Ch03 <-> AI Standard Channel 3/Value
//     Standard Inputs/GVL_IO.AI_LRS_EB1Ch04 <-> AI Standard Channel 4/Value
//   PLC_LMP_VAC_current/PLC_LMP_VAC_current Instance <-> LAMP Fieldbus (EtherCAT)/LRS-EB2 (EP3174-0002)
//     Standard Inputs/GVL_IO.AI_LRS_EB2Ch01 <-> AI Standard Channel 1/Value
//     Standard Inputs/GVL_IO.AI_LRS_EB2Ch02 <-> AI Standard Channel 2/Value
//     Standard Inputs/GVL_IO.AI_LRS_EB2Ch03 <-> AI Standard Channel 3/Value
//     Standard Inputs/GVL_IO.AI_LRS_EB2Ch04 <-> AI Standard Channel 4/Value
//   PLC_LMP_VAC_current/PLC_LMP_VAC_current Instance <-> LAMP Fieldbus (EtherCAT)/LRS-EB3 (EP2339-0021)
//     Standard Inputs/GVL_IO.DiscIO_LRS_EB3Ch02 <-> Channel 2/Input
//     Standard Inputs/GVL_IO.DiscIO_LRS_EB3Ch03 <-> Channel 3/Input
//     Standard Inputs/GVL_IO.DiscIO_LRS_EB3Ch05 <-> Channel 5/Input
//     Standard Inputs/GVL_IO.DiscIO_LRS_EB3Ch06 <-> Channel 6/Input
//     Standard Inputs/GVL_IO.DiscIO_LRS_EB3Ch08 <-> Channel 8/Input
//     Standard Inputs/GVL_IO.DiscIO_LRS_EB3Ch09 <-> Channel 9/Input
//     Standard Inputs/GVL_IO.DiscIO_LRS_EB3Ch11 <-> Channel 11/Input
//     Standard Inputs/GVL_IO.DiscIO_LRS_EB3Ch12 <-> Channel 12/Input
//     Standard Inputs/GVL_IO.DiscIO_LRS_EB3Ch14 <-> Channel 14/Input
//     Standard Inputs/GVL_IO.DiscIO_LRS_EB3Ch15 <-> Channel 15/Input
//     Standard Inputs/GVL_IO.DiscIO_LRS_EB3Ch16 <-> Channel 16/Input
//     Standard Outputs/GVL_IO.DiscIO_LRS_EB3Ch01 <-> Channel 17/Output
//     Standard Outputs/GVL_IO.DiscIO_LRS_EB3Ch04 <-> Channel 20/Output
//     Standard Outputs/GVL_IO.DiscIO_LRS_EB3Ch07 <-> Channel 23/Output
//     Standard Outputs/GVL_IO.DiscIO_LRS_EB3Ch10 <-> Channel 26/Output
//     Standard Outputs/GVL_IO.DiscIO_LRS_EB3Ch13 <-> Channel 29/Output
//   PLC_LMP_VAC_current/PLC_LMP_VAC_current Instance <-> LAMP Fieldbus (EtherCAT)/LRS-EB4 (EP2339-0021)
//     Standard Inputs/GVL_IO.DiscIO_LRS_EB4Ch02 <-> Channel 2/Input
//     Standard Inputs/GVL_IO.DiscIO_LRS_EB4Ch03 <-> Channel 3/Input
//     Standard Inputs/GVL_IO.DiscIO_LRS_EB4Ch05 <-> Channel 5/Input
//     Standard Inputs/GVL_IO.DiscIO_LRS_EB4Ch06 <-> Channel 6/Input
//     Standard Inputs/GVL_IO.DiscIO_LRS_EB4Ch08 <-> Channel 8/Input
//     Standard Inputs/GVL_IO.DiscIO_LRS_EB4Ch09 <-> Channel 9/Input
//     Standard Inputs/GVL_IO.DiscIO_LRS_EB4Ch11 <-> Channel 11/Input
//     Standard Inputs/GVL_IO.DiscIO_LRS_EB4Ch12 <-> Channel 12/Input
//     Standard Inputs/GVL_IO.DiscIO_LRS_EB4Ch14 <-> Channel 14/Input
//     Standard Inputs/GVL_IO.DiscIO_LRS_EB4Ch15 <-> Channel 15/Input
//     Standard Inputs/GVL_IO.DiscIO_LRS_EB4Ch16 <-> Channel 16/Input
//     Standard Outputs/GVL_IO.DiscIO_LRS_EB4Ch01 <-> Channel 17/Output
//     Standard Outputs/GVL_IO.DiscIO_LRS_EB4Ch04 <-> Channel 20/Output
//     Standard Outputs/GVL_IO.DiscIO_LRS_EB4Ch07 <-> Channel 23/Output
//     Standard Outputs/GVL_IO.DiscIO_LRS_EB4Ch10 <-> Channel 26/Output
//     Standard Outputs/GVL_IO.DiscIO_LRS_EB4Ch13 <-> Channel 29/Output
//   PLC_LMP_VAC_current/PLC_LMP_VAC_current Instance <-> LAMP Fieldbus (EtherCAT)/R10_A (EP6002-0002)
//     SerialIO Inputs/GVL_SerialIO.R10_A_P1_stComIn/D[0] <-> COM TxPDO-Map Inputs Channel 1/Data In 0
//     SerialIO Inputs/GVL_SerialIO.R10_A_P1_stComIn/D[10] <-> COM TxPDO-Map Inputs Channel 1/Data In 10
//     SerialIO Inputs/GVL_SerialIO.R10_A_P1_stComIn/D[11] <-> COM TxPDO-Map Inputs Channel 1/Data In 11
//     SerialIO Inputs/GVL_SerialIO.R10_A_P1_stComIn/D[12] <-> COM TxPDO-Map Inputs Channel 1/Data In 12
//     SerialIO Inputs/GVL_SerialIO.R10_A_P1_stComIn/D[13] <-> COM TxPDO-Map Inputs Channel 1/Data In 13
//     SerialIO Inputs/GVL_SerialIO.R10_A_P1_stComIn/D[14] <-> COM TxPDO-Map Inputs Channel 1/Data In 14
//     SerialIO Inputs/GVL_SerialIO.R10_A_P1_stComIn/D[15] <-> COM TxPDO-Map Inputs Channel 1/Data In 15
//     SerialIO Inputs/GVL_SerialIO.R10_A_P1_stComIn/D[16] <-> COM TxPDO-Map Inputs Channel 1/Data In 16
//     SerialIO Inputs/GVL_SerialIO.R10_A_P1_stComIn/D[17] <-> COM TxPDO-Map Inputs Channel 1/Data In 17
//     SerialIO Inputs/GVL_SerialIO.R10_A_P1_stComIn/D[18] <-> COM TxPDO-Map Inputs Channel 1/Data In 18
//     SerialIO Inputs/GVL_SerialIO.R10_A_P1_stComIn/D[19] <-> COM TxPDO-Map Inputs Channel 1/Data In 19
//     SerialIO Inputs/GVL_SerialIO.R10_A_P1_stComIn/D[1] <-> COM TxPDO-Map Inputs Channel 1/Data In 1
//     SerialIO Inputs/GVL_SerialIO.R10_A_P1_stComIn/D[20] <-> COM TxPDO-Map Inputs Channel 1/Data In 20
//     SerialIO Inputs/GVL_SerialIO.R10_A_P1_stComIn/D[21] <-> COM TxPDO-Map Inputs Channel 1/Data In 21
//     SerialIO Inputs/GVL_SerialIO.R10_A_P1_stComIn/D[2] <-> COM TxPDO-Map Inputs Channel 1/Data In 2
//     SerialIO Inputs/GVL_SerialIO.R10_A_P1_stComIn/D[3] <-> COM TxPDO-Map Inputs Channel 1/Data In 3
//     SerialIO Inputs/GVL_SerialIO.R10_A_P1_stComIn/D[4] <-> COM TxPDO-Map Inputs Channel 1/Data In 4
//     SerialIO Inputs/GVL_SerialIO.R10_A_P1_stComIn/D[5] <-> COM TxPDO-Map Inputs Channel 1/Data In 5
//     SerialIO Inputs/GVL_SerialIO.R10_A_P1_stComIn/D[6] <-> COM TxPDO-Map Inputs Channel 1/Data In 6
//     SerialIO Inputs/GVL_SerialIO.R10_A_P1_stComIn/D[7] <-> COM TxPDO-Map Inputs Channel 1/Data In 7
//     SerialIO Inputs/GVL_SerialIO.R10_A_P1_stComIn/D[8] <-> COM TxPDO-Map Inputs Channel 1/Data In 8
//     SerialIO Inputs/GVL_SerialIO.R10_A_P1_stComIn/D[9] <-> COM TxPDO-Map Inputs Channel 1/Data In 9
//     SerialIO Inputs/GVL_SerialIO.R10_A_P2_stComIn/D[0] <-> COM TxPDO-Map Inputs Channel 2/Data In 0
//     SerialIO Inputs/GVL_SerialIO.R10_A_P2_stComIn/D[10] <-> COM TxPDO-Map Inputs Channel 2/Data In 10
//     SerialIO Inputs/GVL_SerialIO.R10_A_P2_stComIn/D[11] <-> COM TxPDO-Map Inputs Channel 2/Data In 11
//     SerialIO Inputs/GVL_SerialIO.R10_A_P2_stComIn/D[12] <-> COM TxPDO-Map Inputs Channel 2/Data In 12
//     SerialIO Inputs/GVL_SerialIO.R10_A_P2_stComIn/D[13] <-> COM TxPDO-Map Inputs Channel 2/Data In 13
//     SerialIO Inputs/GVL_SerialIO.R10_A_P2_stComIn/D[14] <-> COM TxPDO-Map Inputs Channel 2/Data In 14
//     SerialIO Inputs/GVL_SerialIO.R10_A_P2_stComIn/D[15] <-> COM TxPDO-Map Inputs Channel 2/Data In 15
//     SerialIO Inputs/GVL_SerialIO.R10_A_P2_stComIn/D[16] <-> COM TxPDO-Map Inputs Channel 2/Data In 16
//     SerialIO Inputs/GVL_SerialIO.R10_A_P2_stComIn/D[17] <-> COM TxPDO-Map Inputs Channel 2/Data In 17
//     SerialIO Inputs/GVL_SerialIO.R10_A_P2_stComIn/D[18] <-> COM TxPDO-Map Inputs Channel 2/Data In 18
//     SerialIO Inputs/GVL_SerialIO.R10_A_P2_stComIn/D[19] <-> COM TxPDO-Map Inputs Channel 2/Data In 19
//     SerialIO Inputs/GVL_SerialIO.R10_A_P2_stComIn/D[1] <-> COM TxPDO-Map Inputs Channel 2/Data In 1
//     SerialIO Inputs/GVL_SerialIO.R10_A_P2_stComIn/D[20] <-> COM TxPDO-Map Inputs Channel 2/Data In 20
//     SerialIO Inputs/GVL_SerialIO.R10_A_P2_stComIn/D[21] <-> COM TxPDO-Map Inputs Channel 2/Data In 21
//     SerialIO Inputs/GVL_SerialIO.R10_A_P2_stComIn/D[2] <-> COM TxPDO-Map Inputs Channel 2/Data In 2
//     SerialIO Inputs/GVL_SerialIO.R10_A_P2_stComIn/D[3] <-> COM TxPDO-Map Inputs Channel 2/Data In 3
//     SerialIO Inputs/GVL_SerialIO.R10_A_P2_stComIn/D[4] <-> COM TxPDO-Map Inputs Channel 2/Data In 4
//     SerialIO Inputs/GVL_SerialIO.R10_A_P2_stComIn/D[5] <-> COM TxPDO-Map Inputs Channel 2/Data In 5
//     SerialIO Inputs/GVL_SerialIO.R10_A_P2_stComIn/D[6] <-> COM TxPDO-Map Inputs Channel 2/Data In 6
//     SerialIO Inputs/GVL_SerialIO.R10_A_P2_stComIn/D[7] <-> COM TxPDO-Map Inputs Channel 2/Data In 7
//     SerialIO Inputs/GVL_SerialIO.R10_A_P2_stComIn/D[8] <-> COM TxPDO-Map Inputs Channel 2/Data In 8
//     SerialIO Inputs/GVL_SerialIO.R10_A_P2_stComIn/D[9] <-> COM TxPDO-Map Inputs Channel 2/Data In 9
//     SerialIO Inputs/GVL_SerialIO.R10_A_P1_stComIn/Status <-> COM TxPDO-Map Inputs Channel 1/Status
//     SerialIO Inputs/GVL_SerialIO.R10_A_P2_stComIn/Status <-> COM TxPDO-Map Inputs Channel 2/Status
//     SerialIO Outputs/GVL_SerialIO.R10_A_P1_stComOut/Ctrl <-> COM RxPDO-Map Outputs Channel 1/Ctrl
//     SerialIO Outputs/GVL_SerialIO.R10_A_P2_stComOut/Ctrl <-> COM RxPDO-Map Outputs Channel 2/Ctrl
//     SerialIO Outputs/GVL_SerialIO.R10_A_P1_stComOut/D[0] <-> COM RxPDO-Map Outputs Channel 1/Data Out 0
//     SerialIO Outputs/GVL_SerialIO.R10_A_P1_stComOut/D[10] <-> COM RxPDO-Map Outputs Channel 1/Data Out 10
//     SerialIO Outputs/GVL_SerialIO.R10_A_P1_stComOut/D[11] <-> COM RxPDO-Map Outputs Channel 1/Data Out 11
//     SerialIO Outputs/GVL_SerialIO.R10_A_P1_stComOut/D[12] <-> COM RxPDO-Map Outputs Channel 1/Data Out 12
//     SerialIO Outputs/GVL_SerialIO.R10_A_P1_stComOut/D[13] <-> COM RxPDO-Map Outputs Channel 1/Data Out 13
//     SerialIO Outputs/GVL_SerialIO.R10_A_P1_stComOut/D[14] <-> COM RxPDO-Map Outputs Channel 1/Data Out 14
//     SerialIO Outputs/GVL_SerialIO.R10_A_P1_stComOut/D[15] <-> COM RxPDO-Map Outputs Channel 1/Data Out 15
//     SerialIO Outputs/GVL_SerialIO.R10_A_P1_stComOut/D[16] <-> COM RxPDO-Map Outputs Channel 1/Data Out 16
//     SerialIO Outputs/GVL_SerialIO.R10_A_P1_stComOut/D[17] <-> COM RxPDO-Map Outputs Channel 1/Data Out 17
//     SerialIO Outputs/GVL_SerialIO.R10_A_P1_stComOut/D[18] <-> COM RxPDO-Map Outputs Channel 1/Data Out 18
//     SerialIO Outputs/GVL_SerialIO.R10_A_P1_stComOut/D[19] <-> COM RxPDO-Map Outputs Channel 1/Data Out 19
//     SerialIO Outputs/GVL_SerialIO.R10_A_P1_stComOut/D[1] <-> COM RxPDO-Map Outputs Channel 1/Data Out 1
//     SerialIO Outputs/GVL_SerialIO.R10_A_P1_stComOut/D[20] <-> COM RxPDO-Map Outputs Channel 1/Data Out 20
//     SerialIO Outputs/GVL_SerialIO.R10_A_P1_stComOut/D[21] <-> COM RxPDO-Map Outputs Channel 1/Data Out 21
//     SerialIO Outputs/GVL_SerialIO.R10_A_P1_stComOut/D[2] <-> COM RxPDO-Map Outputs Channel 1/Data Out 2
//     SerialIO Outputs/GVL_SerialIO.R10_A_P1_stComOut/D[3] <-> COM RxPDO-Map Outputs Channel 1/Data Out 3
//     SerialIO Outputs/GVL_SerialIO.R10_A_P1_stComOut/D[4] <-> COM RxPDO-Map Outputs Channel 1/Data Out 4
//     SerialIO Outputs/GVL_SerialIO.R10_A_P1_stComOut/D[5] <-> COM RxPDO-Map Outputs Channel 1/Data Out 5
//     SerialIO Outputs/GVL_SerialIO.R10_A_P1_stComOut/D[6] <-> COM RxPDO-Map Outputs Channel 1/Data Out 6
//     SerialIO Outputs/GVL_SerialIO.R10_A_P1_stComOut/D[7] <-> COM RxPDO-Map Outputs Channel 1/Data Out 7
//     SerialIO Outputs/GVL_SerialIO.R10_A_P1_stComOut/D[8] <-> COM RxPDO-Map Outputs Channel 1/Data Out 8
//     SerialIO Outputs/GVL_SerialIO.R10_A_P1_stComOut/D[9] <-> COM RxPDO-Map Outputs Channel 1/Data Out 9
//     SerialIO Outputs/GVL_SerialIO.R10_A_P2_stComOut/D[0] <-> COM RxPDO-Map Outputs Channel 2/Data Out 0
//     SerialIO Outputs/GVL_SerialIO.R10_A_P2_stComOut/D[10] <-> COM RxPDO-Map Outputs Channel 2/Data Out 10
//     SerialIO Outputs/GVL_SerialIO.R10_A_P2_stComOut/D[11] <-> COM RxPDO-Map Outputs Channel 2/Data Out 11
//     SerialIO Outputs/GVL_SerialIO.R10_A_P2_stComOut/D[12] <-> COM RxPDO-Map Outputs Channel 2/Data Out 12
//     SerialIO Outputs/GVL_SerialIO.R10_A_P2_stComOut/D[13] <-> COM RxPDO-Map Outputs Channel 2/Data Out 13
//     SerialIO Outputs/GVL_SerialIO.R10_A_P2_stComOut/D[14] <-> COM RxPDO-Map Outputs Channel 2/Data Out 14
//     SerialIO Outputs/GVL_SerialIO.R10_A_P2_stComOut/D[15] <-> COM RxPDO-Map Outputs Channel 2/Data Out 15
//     SerialIO Outputs/GVL_SerialIO.R10_A_P2_stComOut/D[16] <-> COM RxPDO-Map Outputs Channel 2/Data Out 16
//     SerialIO Outputs/GVL_SerialIO.R10_A_P2_stComOut/D[17] <-> COM RxPDO-Map Outputs Channel 2/Data Out 17
//     SerialIO Outputs/GVL_SerialIO.R10_A_P2_stComOut/D[18] <-> COM RxPDO-Map Outputs Channel 2/Data Out 18
//     SerialIO Outputs/GVL_SerialIO.R10_A_P2_stComOut/D[19] <-> COM RxPDO-Map Outputs Channel 2/Data Out 19
//     SerialIO Outputs/GVL_SerialIO.R10_A_P2_stComOut/D[1] <-> COM RxPDO-Map Outputs Channel 2/Data Out 1
//     SerialIO Outputs/GVL_SerialIO.R10_A_P2_stComOut/D[20] <-> COM RxPDO-Map Outputs Channel 2/Data Out 20
//     SerialIO Outputs/GVL_SerialIO.R10_A_P2_stComOut/D[21] <-> COM RxPDO-Map Outputs Channel 2/Data Out 21
//     SerialIO Outputs/GVL_SerialIO.R10_A_P2_stComOut/D[2] <-> COM RxPDO-Map Outputs Channel 2/Data Out 2
//     SerialIO Outputs/GVL_SerialIO.R10_A_P2_stComOut/D[3] <-> COM RxPDO-Map Outputs Channel 2/Data Out 3
//     SerialIO Outputs/GVL_SerialIO.R10_A_P2_stComOut/D[4] <-> COM RxPDO-Map Outputs Channel 2/Data Out 4
//     SerialIO Outputs/GVL_SerialIO.R10_A_P2_stComOut/D[5] <-> COM RxPDO-Map Outputs Channel 2/Data Out 5
//     SerialIO Outputs/GVL_SerialIO.R10_A_P2_stComOut/D[6] <-> COM RxPDO-Map Outputs Channel 2/Data Out 6
//     SerialIO Outputs/GVL_SerialIO.R10_A_P2_stComOut/D[7] <-> COM RxPDO-Map Outputs Channel 2/Data Out 7
//     SerialIO Outputs/GVL_SerialIO.R10_A_P2_stComOut/D[8] <-> COM RxPDO-Map Outputs Channel 2/Data Out 8
//     SerialIO Outputs/GVL_SerialIO.R10_A_P2_stComOut/D[9] <-> COM RxPDO-Map Outputs Channel 2/Data Out 9
//   PLC_LMP_VAC_current/PLC_LMP_VAC_current Instance <-> LAMP Fieldbus (EtherCAT)/R10_B (EP6002-0002)
//     SerialIO Inputs/GVL_SerialIO.R10_B_P1_stComIn/D[0] <-> COM TxPDO-Map Inputs Channel 1/Data In 0
//     SerialIO Inputs/GVL_SerialIO.R10_B_P1_stComIn/D[10] <-> COM TxPDO-Map Inputs Channel 1/Data In 10
//     SerialIO Inputs/GVL_SerialIO.R10_B_P1_stComIn/D[11] <-> COM TxPDO-Map Inputs Channel 1/Data In 11
//     SerialIO Inputs/GVL_SerialIO.R10_B_P1_stComIn/D[12] <-> COM TxPDO-Map Inputs Channel 1/Data In 12
//     SerialIO Inputs/GVL_SerialIO.R10_B_P1_stComIn/D[13] <-> COM TxPDO-Map Inputs Channel 1/Data In 13
//     SerialIO Inputs/GVL_SerialIO.R10_B_P1_stComIn/D[14] <-> COM TxPDO-Map Inputs Channel 1/Data In 14
//     SerialIO Inputs/GVL_SerialIO.R10_B_P1_stComIn/D[15] <-> COM TxPDO-Map Inputs Channel 1/Data In 15
//     SerialIO Inputs/GVL_SerialIO.R10_B_P1_stComIn/D[16] <-> COM TxPDO-Map Inputs Channel 1/Data In 16
//     SerialIO Inputs/GVL_SerialIO.R10_B_P1_stComIn/D[17] <-> COM TxPDO-Map Inputs Channel 1/Data In 17
//     SerialIO Inputs/GVL_SerialIO.R10_B_P1_stComIn/D[18] <-> COM TxPDO-Map Inputs Channel 1/Data In 18
//     SerialIO Inputs/GVL_SerialIO.R10_B_P1_stComIn/D[19] <-> COM TxPDO-Map Inputs Channel 1/Data In 19
//     SerialIO Inputs/GVL_SerialIO.R10_B_P1_stComIn/D[1] <-> COM TxPDO-Map Inputs Channel 1/Data In 1
//     SerialIO Inputs/GVL_SerialIO.R10_B_P1_stComIn/D[20] <-> COM TxPDO-Map Inputs Channel 1/Data In 20
//     SerialIO Inputs/GVL_SerialIO.R10_B_P1_stComIn/D[21] <-> COM TxPDO-Map Inputs Channel 1/Data In 21
//     SerialIO Inputs/GVL_SerialIO.R10_B_P1_stComIn/D[2] <-> COM TxPDO-Map Inputs Channel 1/Data In 2
//     SerialIO Inputs/GVL_SerialIO.R10_B_P1_stComIn/D[3] <-> COM TxPDO-Map Inputs Channel 1/Data In 3
//     SerialIO Inputs/GVL_SerialIO.R10_B_P1_stComIn/D[4] <-> COM TxPDO-Map Inputs Channel 1/Data In 4
//     SerialIO Inputs/GVL_SerialIO.R10_B_P1_stComIn/D[5] <-> COM TxPDO-Map Inputs Channel 1/Data In 5
//     SerialIO Inputs/GVL_SerialIO.R10_B_P1_stComIn/D[6] <-> COM TxPDO-Map Inputs Channel 1/Data In 6
//     SerialIO Inputs/GVL_SerialIO.R10_B_P1_stComIn/D[7] <-> COM TxPDO-Map Inputs Channel 1/Data In 7
//     SerialIO Inputs/GVL_SerialIO.R10_B_P1_stComIn/D[8] <-> COM TxPDO-Map Inputs Channel 1/Data In 8
//     SerialIO Inputs/GVL_SerialIO.R10_B_P1_stComIn/D[9] <-> COM TxPDO-Map Inputs Channel 1/Data In 9
//     SerialIO Inputs/GVL_SerialIO.R10_B_P2_stComIn/D[0] <-> COM TxPDO-Map Inputs Channel 2/Data In 0
//     SerialIO Inputs/GVL_SerialIO.R10_B_P2_stComIn/D[10] <-> COM TxPDO-Map Inputs Channel 2/Data In 10
//     SerialIO Inputs/GVL_SerialIO.R10_B_P2_stComIn/D[11] <-> COM TxPDO-Map Inputs Channel 2/Data In 11
//     SerialIO Inputs/GVL_SerialIO.R10_B_P2_stComIn/D[12] <-> COM TxPDO-Map Inputs Channel 2/Data In 12
//     SerialIO Inputs/GVL_SerialIO.R10_B_P2_stComIn/D[13] <-> COM TxPDO-Map Inputs Channel 2/Data In 13
//     SerialIO Inputs/GVL_SerialIO.R10_B_P2_stComIn/D[14] <-> COM TxPDO-Map Inputs Channel 2/Data In 14
//     SerialIO Inputs/GVL_SerialIO.R10_B_P2_stComIn/D[15] <-> COM TxPDO-Map Inputs Channel 2/Data In 15
//     SerialIO Inputs/GVL_SerialIO.R10_B_P2_stComIn/D[16] <-> COM TxPDO-Map Inputs Channel 2/Data In 16
//     SerialIO Inputs/GVL_SerialIO.R10_B_P2_stComIn/D[17] <-> COM TxPDO-Map Inputs Channel 2/Data In 17
//     SerialIO Inputs/GVL_SerialIO.R10_B_P2_stComIn/D[18] <-> COM TxPDO-Map Inputs Channel 2/Data In 18
//     SerialIO Inputs/GVL_SerialIO.R10_B_P2_stComIn/D[19] <-> COM TxPDO-Map Inputs Channel 2/Data In 19
//     SerialIO Inputs/GVL_SerialIO.R10_B_P2_stComIn/D[1] <-> COM TxPDO-Map Inputs Channel 2/Data In 1
//     SerialIO Inputs/GVL_SerialIO.R10_B_P2_stComIn/D[20] <-> COM TxPDO-Map Inputs Channel 2/Data In 20
//     SerialIO Inputs/GVL_SerialIO.R10_B_P2_stComIn/D[21] <-> COM TxPDO-Map Inputs Channel 2/Data In 21
//     SerialIO Inputs/GVL_SerialIO.R10_B_P2_stComIn/D[2] <-> COM TxPDO-Map Inputs Channel 2/Data In 2
//     SerialIO Inputs/GVL_SerialIO.R10_B_P2_stComIn/D[3] <-> COM TxPDO-Map Inputs Channel 2/Data In 3
//     SerialIO Inputs/GVL_SerialIO.R10_B_P2_stComIn/D[4] <-> COM TxPDO-Map Inputs Channel 2/Data In 4
//     SerialIO Inputs/GVL_SerialIO.R10_B_P2_stComIn/D[5] <-> COM TxPDO-Map Inputs Channel 2/Data In 5
//     SerialIO Inputs/GVL_SerialIO.R10_B_P2_stComIn/D[6] <-> COM TxPDO-Map Inputs Channel 2/Data In 6
//     SerialIO Inputs/GVL_SerialIO.R10_B_P2_stComIn/D[7] <-> COM TxPDO-Map Inputs Channel 2/Data In 7
//     SerialIO Inputs/GVL_SerialIO.R10_B_P2_stComIn/D[8] <-> COM TxPDO-Map Inputs Channel 2/Data In 8
//     SerialIO Inputs/GVL_SerialIO.R10_B_P2_stComIn/D[9] <-> COM TxPDO-Map Inputs Channel 2/Data In 9
//     SerialIO Inputs/GVL_SerialIO.R10_B_P1_stComIn/Status <-> COM TxPDO-Map Inputs Channel 1/Status
//     SerialIO Inputs/GVL_SerialIO.R10_B_P2_stComIn/Status <-> COM TxPDO-Map Inputs Channel 2/Status
//     SerialIO Outputs/GVL_SerialIO.R10_B_P1_stComOut/Ctrl <-> COM RxPDO-Map Outputs Channel 1/Ctrl
//     SerialIO Outputs/GVL_SerialIO.R10_B_P2_stComOut/Ctrl <-> COM RxPDO-Map Outputs Channel 2/Ctrl
//     SerialIO Outputs/GVL_SerialIO.R10_B_P1_stComOut/D[0] <-> COM RxPDO-Map Outputs Channel 1/Data Out 0
//     SerialIO Outputs/GVL_SerialIO.R10_B_P1_stComOut/D[10] <-> COM RxPDO-Map Outputs Channel 1/Data Out 10
//     SerialIO Outputs/GVL_SerialIO.R10_B_P1_stComOut/D[11] <-> COM RxPDO-Map Outputs Channel 1/Data Out 11
//     SerialIO Outputs/GVL_SerialIO.R10_B_P1_stComOut/D[12] <-> COM RxPDO-Map Outputs Channel 1/Data Out 12
//     SerialIO Outputs/GVL_SerialIO.R10_B_P1_stComOut/D[13] <-> COM RxPDO-Map Outputs Channel 1/Data Out 13
//     SerialIO Outputs/GVL_SerialIO.R10_B_P1_stComOut/D[14] <-> COM RxPDO-Map Outputs Channel 1/Data Out 14
//     SerialIO Outputs/GVL_SerialIO.R10_B_P1_stComOut/D[15] <-> COM RxPDO-Map Outputs Channel 1/Data Out 15
//     SerialIO Outputs/GVL_SerialIO.R10_B_P1_stComOut/D[16] <-> COM RxPDO-Map Outputs Channel 1/Data Out 16
//     SerialIO Outputs/GVL_SerialIO.R10_B_P1_stComOut/D[17] <-> COM RxPDO-Map Outputs Channel 1/Data Out 17
//     SerialIO Outputs/GVL_SerialIO.R10_B_P1_stComOut/D[18] <-> COM RxPDO-Map Outputs Channel 1/Data Out 18
//     SerialIO Outputs/GVL_SerialIO.R10_B_P1_stComOut/D[19] <-> COM RxPDO-Map Outputs Channel 1/Data Out 19
//     SerialIO Outputs/GVL_SerialIO.R10_B_P1_stComOut/D[1] <-> COM RxPDO-Map Outputs Channel 1/Data Out 1
//     SerialIO Outputs/GVL_SerialIO.R10_B_P1_stComOut/D[20] <-> COM RxPDO-Map Outputs Channel 1/Data Out 20
//     SerialIO Outputs/GVL_SerialIO.R10_B_P1_stComOut/D[21] <-> COM RxPDO-Map Outputs Channel 1/Data Out 21
//     SerialIO Outputs/GVL_SerialIO.R10_B_P1_stComOut/D[2] <-> COM RxPDO-Map Outputs Channel 1/Data Out 2
//     SerialIO Outputs/GVL_SerialIO.R10_B_P1_stComOut/D[3] <-> COM RxPDO-Map Outputs Channel 1/Data Out 3
//     SerialIO Outputs/GVL_SerialIO.R10_B_P1_stComOut/D[4] <-> COM RxPDO-Map Outputs Channel 1/Data Out 4
//     SerialIO Outputs/GVL_SerialIO.R10_B_P1_stComOut/D[5] <-> COM RxPDO-Map Outputs Channel 1/Data Out 5
//     SerialIO Outputs/GVL_SerialIO.R10_B_P1_stComOut/D[6] <-> COM RxPDO-Map Outputs Channel 1/Data Out 6
//     SerialIO Outputs/GVL_SerialIO.R10_B_P1_stComOut/D[7] <-> COM RxPDO-Map Outputs Channel 1/Data Out 7
//     SerialIO Outputs/GVL_SerialIO.R10_B_P1_stComOut/D[8] <-> COM RxPDO-Map Outputs Channel 1/Data Out 8
//     SerialIO Outputs/GVL_SerialIO.R10_B_P1_stComOut/D[9] <-> COM RxPDO-Map Outputs Channel 1/Data Out 9
//     SerialIO Outputs/GVL_SerialIO.R10_B_P2_stComOut/D[0] <-> COM RxPDO-Map Outputs Channel 2/Data Out 0
//     SerialIO Outputs/GVL_SerialIO.R10_B_P2_stComOut/D[10] <-> COM RxPDO-Map Outputs Channel 2/Data Out 10
//     SerialIO Outputs/GVL_SerialIO.R10_B_P2_stComOut/D[11] <-> COM RxPDO-Map Outputs Channel 2/Data Out 11
//     SerialIO Outputs/GVL_SerialIO.R10_B_P2_stComOut/D[12] <-> COM RxPDO-Map Outputs Channel 2/Data Out 12
//     SerialIO Outputs/GVL_SerialIO.R10_B_P2_stComOut/D[13] <-> COM RxPDO-Map Outputs Channel 2/Data Out 13
//     SerialIO Outputs/GVL_SerialIO.R10_B_P2_stComOut/D[14] <-> COM RxPDO-Map Outputs Channel 2/Data Out 14
//     SerialIO Outputs/GVL_SerialIO.R10_B_P2_stComOut/D[15] <-> COM RxPDO-Map Outputs Channel 2/Data Out 15
//     SerialIO Outputs/GVL_SerialIO.R10_B_P2_stComOut/D[16] <-> COM RxPDO-Map Outputs Channel 2/Data Out 16
//     SerialIO Outputs/GVL_SerialIO.R10_B_P2_stComOut/D[17] <-> COM RxPDO-Map Outputs Channel 2/Data Out 17
//     SerialIO Outputs/GVL_SerialIO.R10_B_P2_stComOut/D[18] <-> COM RxPDO-Map Outputs Channel 2/Data Out 18
//     SerialIO Outputs/GVL_SerialIO.R10_B_P2_stComOut/D[19] <-> COM RxPDO-Map Outputs Channel 2/Data Out 19
//     SerialIO Outputs/GVL_SerialIO.R10_B_P2_stComOut/D[1] <-> COM RxPDO-Map Outputs Channel 2/Data Out 1
//     SerialIO Outputs/GVL_SerialIO.R10_B_P2_stComOut/D[20] <-> COM RxPDO-Map Outputs Channel 2/Data Out 20
//     SerialIO Outputs/GVL_SerialIO.R10_B_P2_stComOut/D[21] <-> COM RxPDO-Map Outputs Channel 2/Data Out 21
//     SerialIO Outputs/GVL_SerialIO.R10_B_P2_stComOut/D[2] <-> COM RxPDO-Map Outputs Channel 2/Data Out 2
//     SerialIO Outputs/GVL_SerialIO.R10_B_P2_stComOut/D[3] <-> COM RxPDO-Map Outputs Channel 2/Data Out 3
//     SerialIO Outputs/GVL_SerialIO.R10_B_P2_stComOut/D[4] <-> COM RxPDO-Map Outputs Channel 2/Data Out 4
//     SerialIO Outputs/GVL_SerialIO.R10_B_P2_stComOut/D[5] <-> COM RxPDO-Map Outputs Channel 2/Data Out 5
//     SerialIO Outputs/GVL_SerialIO.R10_B_P2_stComOut/D[6] <-> COM RxPDO-Map Outputs Channel 2/Data Out 6
//     SerialIO Outputs/GVL_SerialIO.R10_B_P2_stComOut/D[7] <-> COM RxPDO-Map Outputs Channel 2/Data Out 7
//     SerialIO Outputs/GVL_SerialIO.R10_B_P2_stComOut/D[8] <-> COM RxPDO-Map Outputs Channel 2/Data Out 8
//     SerialIO Outputs/GVL_SerialIO.R10_B_P2_stComOut/D[9] <-> COM RxPDO-Map Outputs Channel 2/Data Out 9
//   PLC_LMP_VAC_current/PLC_LMP_VAC_current Instance <-> LAMP Fieldbus (EtherCAT)/Term 1 (EK1200)/Term 2 (EL3064)
//     Standard Inputs/GVL_IO.AI_Term2_Ch{1..4} <-> AI Standard Channel {1..4}/Value  (4 links)
//   PLC_LMP_VAC_current/PLC_LMP_VAC_current Instance <-> LAMP Fieldbus (EtherCAT)/Term 1 (EK1200)/Term 3 (EL3064)
//     Standard Inputs/GVL_IO.AI_Term3_Ch{1..4} <-> AI Standard Channel {1..4}/Value  (4 links)
//   PLC_LMP_VAC_current/PLC_LMP_VAC_current Instance <-> LAMP Fieldbus (EtherCAT)/Term 1 (EK1200)/Term 4 (EL1008)
//     Standard Inputs/GVL_IO.DI_Term4_Ch{1..8} <-> Channel {1..8}/Input  (8 links)
//   PLC_LMP_VAC_current/PLC_LMP_VAC_current Instance <-> LAMP Fieldbus (EtherCAT)/Term 1 (EK1200)/Term 5 (EL2008)
//     Standard Outputs/GVL_IO.DO_Term5_Ch{1..8} <-> Channel {1..8}/Output  (8 links)
//   PLC_LMP_VAC_current/PLC_LMP_VAC_current Instance <-> LAMP Fieldbus (EtherCAT)/Term 1 (EK1200)/Term 6 (EL2798)
//     Standard Outputs/GVL_IO.DO_Term6_Ch{1..8} <-> Channel {1..8}/Output  (8 links)
//   PLC_LMP_VAC_current/PLC_LMP_VAC_current Instance <-> LAMP(EtherCAT Slave)
//     Standard Inputs/GVL_IO.LAMP_BRB_{1..8} <-> Inputs/i_xAux_{1..8}  (8 links)
//     Standard Inputs/GVL_IO.i_rAuxVG{1..4} <-> Inputs/i_rAuxVG_{1..4}  (4 links)
//     Standard Outputs/GVL_IO.LAMP_BCO_{1..8} <-> Outputs/q_xAux_{1..8}  (8 links)
//     Standard Outputs/GVL_IO.LAMP_MPS_{1..8} <-> Outputs/q_xMPS_{1..8}  (8 links)
//     Standard Outputs/GVL_IO.q_rLampAuxVG{1..4} <-> Outputs/q_rAuxVG{1..4}  (4 links)

CONFIGURATION PLC_LMP_VAC_current
    RESOURCE PLC ON TwinCAT3
        TASK Standard(INTERVAL := T#10ms, PRIORITY := 8);
        TASK SerialIO(INTERVAL := T#5ms, PRIORITY := 6);
        PROGRAM MAIN WITH Standard : MAIN;
        PROGRAM P_Serial_Com WITH SerialIO : P_Serial_Com;
    END_RESOURCE
END_CONFIGURATION

// ---- Global Variables/GVL.TcGVL
VAR_GLOBAL
	(* User Memory Variables *)

	LMP_Sys00	: System_Struct;
	xLOTO: BOOL := TRUE;
	g_rExtIlkPres: REAL; //User-specified pressure for ext. interlocking
	g_iExtIlkGauge: INT; //User-specified gauge to interlock from
	g_xExtIlkRO: BOOL := FALSE; //LAMP ext. interlock output
	g_iActivePfeiffers : INT := 10;
	
	g_xPTMGroupRun: ARRAY [0..10] OF BOOL;
	
	(* Modbus TCP *)
   	mb_Input_Coils       				: ARRAY [0..255] OF BOOL; 	(* test mb_Input_Coils[0] with "modpoll -r 32769 -t 1 127.0.0.1" *)
    mb_Output_Coils      				: ARRAY [0..255] OF BOOL;	(* test mb_Output_Coils[0] with "modpoll -r 32769 -t 0 127.0.0.1" *)
	mb_Input_Registers 				: ARRAY [0..255] OF WORD; 	(* test mb_Input_Registers[0] with "modpoll -r 32769 -t 3 127.0.0.1" *)
	mb_Output_Registers 				: ARRAY [0..255] OF WORD; 	(* test mb_Output_Registers[0] with "modpoll -r 32769 -t 4 127.0.0.1" *)
	mb_PLC_Memory 			AT %MW0 	: ARRAY [0..1000] OF WORD; 	(* test mb_PLC_Memory[0] with "modpoll -r 12289 -t 4 127.0.0.1" *)


END_VAR

// ---- Global Variables/GVL_Autosave.TcGVL
VAR_GLOBAL PERSISTENT
	
gp_LMP_VG			:	ARRAY[0..50] OF ST_VG;


END_VAR

// ---- Global Variables/GVL_COM_Buffers.TcGVL
VAR_GLOBAL
	
	DET_P1_SerialRXBuffer : ComBuffer;
	DET_P1_SerialTXBuffer : ComBuffer;
	
	DET_P2_SerialRXBuffer : ComBuffer;
	DET_P2_SerialTXBuffer : ComBuffer;

	IC_P1_SerialRXBuffer : ComBuffer;
	IC_P1_SerialTXBuffer : ComBuffer;

	IC_P2_SerialRXBuffer : ComBuffer;
	IC_P2_SerialTXBuffer : ComBuffer;

	R10_A_P1_SerialRXBuffer : ComBuffer;
	R10_A_P1_SerialTXBuffer : ComBuffer;
	
	R10_A_P2_SerialRXBuffer : ComBuffer;
	R10_A_P2_SerialTXBuffer : ComBuffer;
	
	R10_B_P1_SerialRXBuffer : ComBuffer;
	R10_B_P1_SerialTXBuffer : ComBuffer;
	
	R10_B_P2_SerialRXBuffer : ComBuffer;
	R10_B_P2_SerialTXBuffer : ComBuffer;
	
END_VAR

// ---- Global Variables/GVL_Devices.TcGVL
VAR_GLOBAL
	
(* Soft IO Variables include switch commands, interlocks and alarms mapped to EPICS *)
	
(* All Pfeiffer Pumps - on Port 1 of the Interaction chamber EP6002 *)
	g_astPfe_CTRL 			: ARRAY[1..20] OF ST_PfeifferControl;
	g_astPfe_RBK 			: ARRAY[1..20] OF ST_PfeifferStatus;
	g_afbPfe_SerialDriver 	: ARRAY[1..20] OF FB_PfeifferSerialDriver;

(* Port 1 of the R10 EB1 Serial Interface (corresponds to LMP_PTM44) *)
	g_astTD20_RBK			: ST_TD20Status;
	g_astTD20_SerialDriver	: FB_TD20SerialDriver;

//Array of Pfeiffer PTM objects...see below
 aLMP_PTM		:	ARRAY[10..41] OF ST_PfeifferPTM;
	
(*
LAMP Pfeiffer PTM EPICS -> RS485 / array mapping (NOTE: RS485 address set in p_Initialize)

Current name	RS485 address	New array name			Pump type
(* Differential pumping *)
LMP_PTM10			1			aLMP_PTM[10]		DP 300L/s
LMP_PTM11			2			aLMP_PTM[11]     	DP 300L/s
(* Interaction Chamber *)
LMP_PTM20			7			aLMP_PTM[20]		IC 300L/s
LMP_PTM21			8			aLMP_PTM[21]	 	IC 400L/s
(* Detector Chamber *)
LMP_PTM30			3			aLMP_PTM[30] 		DET 700L/s
LMP_PTM31			4			aLMP_PTM[31]		DET 700L/s
LMP_PTM32			5			aLMP_PTM[32]		DET 700L/s
LMP_PTM33			6			aLMP_PTM[33]	 	DET 700L/s
(* Gas Jet 1 *)
LMP_PTM40			9			aLMP_PTM[40]	 	GJ 300L/s, TC110
LMP_PTM41			10			aLMP_PTM[41]		GJ 300L/s, TC110
 *)
	LMP_PTM44	:	ST_OerlikonPTM;


(* VGC *)
	LMP_VGC30		:	ST_VGC;
	LMP_VGC10		:	ST_VGC;
	H2E_VGC01		:	ST_VGC;
	H2E_VGC02		:	ST_VGC;

(* VRC *)
	LMP_VRC01		:	ST_VRC;
	LMP_VRC02		:	ST_VRC;
	LMP_VRC03		:	ST_VRC;
	LMP_VRC04		:	ST_VRC;
	LMP_VRC05		:	ST_VRC;
	LMP_VRC06		:	ST_VRC;
	LMP_VRC07		:	ST_VRC;

(* VCC - the simplest kind *)
	LMP_VCCUSR		:	ST_VCC;

(* VG Vacuum Gauges *)
	LMP_GPI_D1		:	ST_VG; (* dummy pirani, there is a difference, see the dumb_gauge function *)

	LMP_VG			:	ARRAY[0..50] OF ST_VG;
	H2E_VG01        :   ST_VG;
	H2E_VG02		:	ST_VG;		

(* Relay Outputs *)

	LMP_RO	:	ARRAY[0..50] OF BOOL;

(* Encoder *)
	LMP_ENC01	:	ST_Encoder;
	LMP_ENC02	:	ST_Encoder;
	LMP_ENC03	:	ST_Encoder;

END_VAR

// ---- Global Variables/GVL_IO.TcGVL
VAR_GLOBAL
	
(* Hardware Input/Output Declaration *)
(* Hardware Inputs & Outputs are mapped to 'Soft' IO tags in the list below. *)
(* There should be one matching IO tag for each physical IO in System Manager. *)
(* IMPORTANT - This list should change only  if physical IO modules are added or removed *)
(* from the PLC. Otherwise, this map and linking should never change. *)

	AI_Term2_Ch1 AT %I* : INT;
	AI_Term2_Ch2 AT %I* : INT;
	AI_Term2_Ch3 AT %I* : INT;
	AI_Term2_Ch4 AT %I* : INT;

	AI_Term3_Ch1 AT %I* : INT;
	AI_Term3_Ch2 AT %I* : INT;
	AI_Term3_Ch3 AT %I* : INT;
	AI_Term3_Ch4 AT %I* : INT;

	DI_Term4_Ch1 AT %I* : BOOL;
	DI_Term4_Ch2 AT %I* : BOOL;
	DI_Term4_Ch3 AT %I* : BOOL;
	DI_Term4_Ch4 AT %I* : BOOL;
	DI_Term4_Ch5 AT %I* : BOOL;
	DI_Term4_Ch6 AT %I* : BOOL;
	DI_Term4_Ch7 AT %I* : BOOL;
	DI_Term4_Ch8 AT %I* : BOOL;

	DO_Term5_Ch1 AT %Q* : BOOL;
	DO_Term5_Ch2 AT %Q* : BOOL;
	DO_Term5_Ch3 AT %Q* : BOOL;
	DO_Term5_Ch4 AT %Q* : BOOL;
	DO_Term5_Ch5 AT %Q* : BOOL;
	DO_Term5_Ch6 AT %Q* : BOOL;
	DO_Term5_Ch7 AT %Q* : BOOL;
	DO_Term5_Ch8 AT %Q* : BOOL;
	
	DO_Term6_Ch1 AT %Q* : BOOL;
	DO_Term6_Ch2 AT %Q* : BOOL;
	DO_Term6_Ch3 AT %Q* : BOOL;
	DO_Term6_Ch4 AT %Q* : BOOL;
	DO_Term6_Ch5 AT %Q* : BOOL;
	DO_Term6_Ch6 AT %Q* : BOOL;
	DO_Term6_Ch7 AT %Q* : BOOL;
	DO_Term6_Ch8 AT %Q* : BOOL;	
	
	(* Fieldbus PLC IO *)
	
(* IC interfaace *)
	
	(*EP3174 *)
	AI_IC_EB2Ch01 AT %I* : INT;
	AI_IC_EB2Ch02 AT %I* : INT;
	AI_IC_EB2Ch03 AT %I* : INT;
	AI_IC_EB2Ch04 AT %I* : INT;
	
	(*EP2624*)
	RelayO_IC_EB3Ch01 AT %Q* : BOOL;
	RelayO_IC_EB3Ch02 AT %Q* : BOOL;
	RelayO_IC_EB3Ch03 AT %Q* : BOOL;
	RelayO_IC_EB3Ch04 AT %Q* : BOOL;
	
	
	(*EP2339*)
	DiscIO_IC_EB4Ch01 AT %Q* : BOOL; (* note, these channels can be configured as input or output*)
	DiscIO_IC_EB4Ch02 AT %I* : BOOL;
	DiscIO_IC_EB4Ch03 AT %I* : BOOL;
	DiscIO_IC_EB4Ch04 AT %Q* : BOOL;
	DiscIO_IC_EB4Ch05 AT %I* : BOOL;
	DiscIO_IC_EB4Ch06 AT %I* : BOOL;
	DiscIO_IC_EB4Ch07 AT %Q* : BOOL;
	DiscIO_IC_EB4Ch08 AT %I* : BOOL;
	DiscIO_IC_EB4Ch09 AT %I* : BOOL;
	DiscIO_IC_EB4Ch10 AT %Q* : BOOL;
	DiscIO_IC_EB4Ch11 AT %I* : BOOL;
	DiscIO_IC_EB4Ch12 AT %I* : BOOL;
	DiscIO_IC_EB4Ch13 AT %Q* : BOOL;
	DiscIO_IC_EB4Ch14 AT %I* : BOOL;
	DiscIO_IC_EB4Ch15 AT %I* : BOOL;
	DiscIO_IC_EB4Ch16 AT %I* : BOOL;
	
(* DET interfaace *)
	
	(*EP3174 *)
	AI_DET_EB2Ch01 AT %I* : INT;
	AI_DET_EB2Ch02 AT %I* : INT;
	AI_DET_EB2Ch03 AT %I* : INT;
	AI_DET_EB2Ch04 AT %I* : INT;
	
	(*EP2624*)
	RelayO_DET_EB3Ch01 AT %Q* : BOOL;
	RelayO_DET_EB3Ch02 AT %Q* : BOOL;
	RelayO_DET_EB3Ch03 AT %Q* : BOOL;
	RelayO_DET_EB3Ch04 AT %Q* : BOOL;
	
	(*EP2339*)
	DiscIO_DET_EB4Ch01 AT %Q* : BOOL; (* note, these channels can be configured as input or output*)
	DiscIO_DET_EB4Ch02 AT %I* : BOOL;
	DiscIO_DET_EB4Ch03 AT %I* : BOOL;
	DiscIO_DET_EB4Ch04 AT %Q* : BOOL;
	DiscIO_DET_EB4Ch05 AT %I* : BOOL;
	DiscIO_DET_EB4Ch06 AT %I* : BOOL;
	DiscIO_DET_EB4Ch07 AT %Q* : BOOL;
	DiscIO_DET_EB4Ch08 AT %I* : BOOL;
	DiscIO_DET_EB4Ch09 AT %I* : BOOL;
	DiscIO_DET_EB4Ch10 AT %Q* : BOOL;
	DiscIO_DET_EB4Ch11 AT %I* : BOOL;
	DiscIO_DET_EB4Ch12 AT %I* : BOOL;
	DiscIO_DET_EB4Ch13 AT %Q* : BOOL;
	DiscIO_DET_EB4Ch14 AT %I* : BOOL;
	DiscIO_DET_EB4Ch15 AT %I* : BOOL;
	DiscIO_DET_EB4Ch16 AT %I* : BOOL;	
	
	(*EP2624*)
	RelayO_DET_EB5Ch01 AT %Q* : BOOL;
	RelayO_DET_EB5Ch02 AT %Q* : BOOL;
	RelayO_DET_EB5Ch03 AT %Q* : BOOL;
	RelayO_DET_EB5Ch04 AT %Q* : BOOL;	
	
	(*EP3174 *)
	AI_DET_EB6Ch01 AT %I* : INT;
	AI_DET_EB6Ch02 AT %I* : INT;
	AI_DET_EB6Ch03 AT %I* : INT;
	AI_DET_EB6Ch04 AT %I* : INT;
	

(* GJ interfaace *)

	(*EP2624*)
	RelayO_GJ_EB1Ch01 AT %Q* : BOOL;
	RelayO_GJ_EB1Ch02 AT %Q* : BOOL;
	RelayO_GJ_EB1Ch03 AT %Q* : BOOL;
	RelayO_GJ_EB1Ch04 AT %Q* : BOOL;
	
	(*EP3174 *)
	AI_GJ_EB2Ch01 AT %I* : INT;
	AI_GJ_EB2Ch02 AT %I* : INT;
	AI_GJ_EB2Ch03 AT %I* : INT;
	AI_GJ_EB2Ch04 AT %I* : INT;
	
	(*EP2339*)
	DiscIO_GJ_EB3Ch01 AT %Q* : BOOL; (* note, these channels can be configured as input or output*)
	DiscIO_GJ_EB3Ch02 AT %I* : BOOL;
	DiscIO_GJ_EB3Ch03 AT %I* : BOOL;
	DiscIO_GJ_EB3Ch04 AT %Q* : BOOL;
	DiscIO_GJ_EB3Ch05 AT %I* : BOOL;
	DiscIO_GJ_EB3Ch06 AT %I* : BOOL;
	DiscIO_GJ_EB3Ch07 AT %Q* : BOOL;
	DiscIO_GJ_EB3Ch08 AT %I* : BOOL;
	DiscIO_GJ_EB3Ch09 AT %I* : BOOL;
	DiscIO_GJ_EB3Ch10 AT %Q* : BOOL;
	DiscIO_GJ_EB3Ch11 AT %I* : BOOL;
	DiscIO_GJ_EB3Ch12 AT %I* : BOOL;
	DiscIO_GJ_EB3Ch13 AT %Q* : BOOL;
	DiscIO_GJ_EB3Ch14 AT %I* : BOOL;
	DiscIO_GJ_EB3Ch15 AT %I* : BOOL;
	DiscIO_GJ_EB3Ch16 AT %I* : BOOL;
	
	(*EP3174 *)
	AI_GJ_EB4Ch01 AT %I* : INT;
	AI_GJ_EB4Ch02 AT %I* : INT;
	AI_GJ_EB4Ch03 AT %I* : INT;
	AI_GJ_EB4Ch04 AT %I* : INT;
	
	
(*  LRS interface  *)
	
	(*EP3174 *)
	AI_LRS_EB1Ch01 AT %I* : INT;
	AI_LRS_EB1Ch02 AT %I* : INT;
	AI_LRS_EB1Ch03 AT %I* : INT;
	AI_LRS_EB1Ch04 AT %I* : INT;
	
	(*EP3174 *)
	AI_LRS_EB2Ch01 AT %I* : INT;
	AI_LRS_EB2Ch02 AT %I* : INT;
	AI_LRS_EB2Ch03 AT %I* : INT;
	AI_LRS_EB2Ch04 AT %I* : INT;
	
	(*EP2339*)	
	DiscIO_LRS_EB3Ch01 AT %Q* : BOOL;(* note, these channels can be configured as input or output*)
	DiscIO_LRS_EB3Ch02 AT %I* : BOOL;
	DiscIO_LRS_EB3Ch03 AT %I* : BOOL;
	DiscIO_LRS_EB3Ch04 AT %Q* : BOOL;
	DiscIO_LRS_EB3Ch05 AT %I* : BOOL;
	DiscIO_LRS_EB3Ch06 AT %I* : BOOL;
	DiscIO_LRS_EB3Ch07 AT %Q* : BOOL;
	DiscIO_LRS_EB3Ch08 AT %I* : BOOL;
	DiscIO_LRS_EB3Ch09 AT %I* : BOOL;
	DiscIO_LRS_EB3Ch10 AT %Q* : BOOL;
	DiscIO_LRS_EB3Ch11 AT %I* : BOOL;
	DiscIO_LRS_EB3Ch12 AT %I* : BOOL;
	DiscIO_LRS_EB3Ch13 AT %Q* : BOOL;
	DiscIO_LRS_EB3Ch14 AT %I* : BOOL;
	DiscIO_LRS_EB3Ch15 AT %I* : BOOL;
	DiscIO_LRS_EB3Ch16 AT %I* : BOOL;
	
	(*EP2339*)
	DiscIO_LRS_EB4Ch01 AT %Q* : BOOL;(* note, these channels can be configured as input or output*)
	DiscIO_LRS_EB4Ch02 AT %I* : BOOL;
	DiscIO_LRS_EB4Ch03 AT %I* : BOOL;
	DiscIO_LRS_EB4Ch04 AT %Q* : BOOL;
	DiscIO_LRS_EB4Ch05 AT %I* : BOOL;
	DiscIO_LRS_EB4Ch06 AT %I* : BOOL;
	DiscIO_LRS_EB4Ch07 AT %Q* : BOOL;
	DiscIO_LRS_EB4Ch08 AT %I* : BOOL;
	DiscIO_LRS_EB4Ch09 AT %I* : BOOL;
	DiscIO_LRS_EB4Ch10 AT %Q* : BOOL;
	DiscIO_LRS_EB4Ch11 AT %I* : BOOL;
	DiscIO_LRS_EB4Ch12 AT %I* : BOOL;
	DiscIO_LRS_EB4Ch13 AT %Q* : BOOL;
	DiscIO_LRS_EB4Ch14 AT %I* : BOOL;
	DiscIO_LRS_EB4Ch15 AT %I* : BOOL;
	DiscIO_LRS_EB4Ch16 AT %I* : BOOL;
	
(* H2E interfaace *)	

	(*EP2339*)
	DiscIO_H2E_EB1Ch01 AT %Q* : BOOL; (* note, these channels can be configured as input or output*)
	DiscIO_H2E_EB1Ch02 AT %I* : BOOL;
	DiscIO_H2E_EB1Ch03 AT %I* : BOOL;
	DiscIO_H2E_EB1Ch04 AT %Q* : BOOL;
	DiscIO_H2E_EB1Ch05 AT %I* : BOOL;
	DiscIO_H2E_EB1Ch06 AT %I* : BOOL;
	DiscIO_H2E_EB1Ch07 AT %Q* : BOOL;
	DiscIO_H2E_EB1Ch08 AT %I* : BOOL;
	DiscIO_H2E_EB1Ch09 AT %I* : BOOL;
	DiscIO_H2E_EB1Ch10 AT %Q* : BOOL;
	DiscIO_H2E_EB1Ch11 AT %I* : BOOL;
	DiscIO_H2E_EB1Ch12 AT %I* : BOOL;
	DiscIO_H2E_EB1Ch13 AT %Q* : BOOL;
	DiscIO_H2E_EB1Ch14 AT %I* : BOOL;
	DiscIO_H2E_EB1Ch15 AT %I* : BOOL;
	DiscIO_H2E_EB1Ch16 AT %I* : BOOL;	
	
	(*EP3174 *)
	AI_H2E_EB2Ch01 AT %I* : INT;
	AI_H2E_EB2Ch02 AT %I* : INT;
	AI_H2E_EB2Ch03 AT %I* : INT;
	AI_H2E_EB2Ch04 AT %I* : INT;

(* MPS Outputs to another PLC (ECAT slave interface) *)
	LAMP_MPS_1 AT %Q*	:	BOOL;
	LAMP_MPS_2 AT %Q*	:	BOOL;
	LAMP_MPS_3 AT %Q*	:	BOOL;
	LAMP_MPS_4 AT %Q*	:	BOOL;
	LAMP_MPS_5 AT %Q*	:	BOOL;
	LAMP_MPS_6 AT %Q*	:	BOOL;
	LAMP_MPS_7 AT %Q*	:	BOOL;
	LAMP_MPS_8 AT %Q*	:	BOOL;

(* Misc Outputs to another PLC (ECAT slave interface) *)

	LAMP_BCO_1 AT %Q*	:	BOOL;
	LAMP_BCO_2 AT %Q*	:	BOOL;
	LAMP_BCO_3 AT %Q*	:	BOOL;
	LAMP_BCO_4 AT %Q*	:	BOOL;
	LAMP_BCO_5 AT %Q*	:	BOOL;
	LAMP_BCO_6 AT %Q*	:	BOOL;
	LAMP_BCO_7 AT %Q*	:	BOOL;
	LAMP_BCO_8 AT %Q*	:	BOOL;

	q_rLampAuxVG1 AT %Q*	:	REAL;
	q_rLampAuxVG2 AT %Q*	:	REAL;
	q_rLampAuxVG3 AT %Q*	:	REAL;
	q_rLampAuxVG4 AT %Q*	:	REAL;

(* Misc Inputs from another PLC (ECAT slave interfaace) *)

	LAMP_BRB_1 AT %I*	:	BOOL;
	LAMP_BRB_2 AT %I*	:	BOOL;
	LAMP_BRB_3 AT %I*	:	BOOL;
	LAMP_BRB_4 AT %I*	:	BOOL;
	LAMP_BRB_5 AT %I*	:	BOOL;
	LAMP_BRB_6 AT %I*	:	BOOL;
	LAMP_BRB_7 AT %I*	:	BOOL;
	LAMP_BRB_8 AT %I*	:	BOOL;

	i_rAuxVG1 AT %I*	:	REAL;
	i_rAuxVG2 AT %I*	:	REAL;
	i_rAuxVG3 AT %I*	:	REAL;
	i_rAuxVG4 AT %I*	:	REAL;
	

END_VAR

// ---- Global Variables/GVL_SerialIO.TcGVL
VAR_GLOBAL
	

	DET_P1_stComIn		AT %I*	:	EL6inData22B (*KL6inData22B*);
	DET_P1_stComOut		AT %Q*	:	EL6outData22B (*KL6outData22B*);

	DET_P2_stComIn		AT %I*	:	EL6inData22B (*KL6inData22B*);
	DET_P2_stComOut		AT %Q*	:	EL6outData22B (*KL6outData22B*);

	IC_P1_stComIn		AT %I*	:	EL6inData22B (*KL6inData22B*);
	IC_P1_stComOut		AT %Q*	:	EL6outData22B (*KL6outData22B*);

	IC_P2_stComIn		AT %I*	:	EL6inData22B (*KL6inData22B*);
	IC_P2_stComOut		AT %Q*	:	EL6outData22B (*KL6outData22B*);

	R10_A_P1_stComIn		AT %I*	:	EL6inData22B (*KL6inData22B*);
	R10_A_P1_stComOut		AT %Q*	:	EL6outData22B (*KL6outData22B*);

	R10_A_P2_stComIn		AT %I*	:	EL6inData22B (*KL6inData22B*);
	R10_A_P2_stComOut		AT %Q*	:	EL6outData22B (*KL6outData22B*);

	R10_B_P1_stComIn		AT %I*	:	EL6inData22B (*KL6inData22B*);
	R10_B_P1_stComOut		AT %Q*	:	EL6outData22B (*KL6outData22B*);

	R10_B_P2_stComIn		AT %I*	:	EL6inData22B (*KL6inData22B*);
	R10_B_P2_stComOut		AT %Q*	:	EL6outData22B (*KL6outData22B*);
	
	
END_VAR

// ---- POUs/MAIN.TcPOU
PROGRAM MAIN
VAR

	fbFSInit : R_TRIG;

	fb_S_UPS	:	FB_S_UPS;
	
END_VAR

(* 	MAIN *)
(* 	For this logic to work properly, program has to execute in the following order after initializaion,
	1. EPICS Rx UPDATE
	2. HARDWIRED I/O UPDATE
	3. RESOLVE LOGIC
	4. EPICS Tx UPDATE
*)
fb_S_UPS(iPLCPort:=851);

(* INITIALIZATION - Make one pass on startup. *)
	fbFSInit(CLK := TRUE,
			  Q => LMP_Sys00.xFirstScan);

	IF LMP_Sys00.xFirstScan THEN p_Initialize(); END_IF;

(* 	EPICS Rx UPDATE
 	Modbus Map Receive - Do not refresh EPICS commands of first pass.
	IMPORTANT: This is the FIRST subroutine TO be called after first-pass initialization. It must run AT the top OF the scan 
*)
	IF NOT LMP_Sys00.xFirstScan THEN p_ModbusMapRx(); END_IF;
p_Autosave();

(* 	HARD-WIRED I/O UPDATE
	Update IO 
*)
p_Serial_PTM_IO();

p_SoftIOMap();



(* 	RESOLVE LOGIC
	DeVRCe Control & Monitoring 
*)
p_PTMSup();
p_GaugeSup();
p_ValveSup();
Encoders();
Ext_Interlocks();


(* 	EPICS Tx UPDATE
	Modbus Map Receive
	IMPORTANT: This is the LAST subroutine to be called. It must run at the bottom of the scan 
*)
p_ModbusMapTx();

END_PROGRAM

// ---- POUs/p_Initialize.TcPOU
PROGRAM p_Initialize
VAR

	catch: INT;
	xFirstScan: BOOL := TRUE;
	counter : INT;
END_VAR

IF xFirstScan THEN
xFirstScan := FALSE;

(* Pfeiffers *)
FOR counter := 1 TO g_iActivePfeiffers DO
	g_astPfe_CTRL[counter].iSerialAddress := counter;
	g_astPfe_CTRL[counter].xEnableComm := TRUE;
END_FOR

	aLMP_PTM[10].iPumpGrp	:= 0;
	aLMP_PTM[10].xActive 	:= 1;	
	aLMP_PTM[11].iPumpGrp	:= 1;
	aLMP_PTM[11].xActive	:= 1;
	aLMP_PTM[20].iPumpGrp	:= 2;
	aLMP_PTM[20].xActive	:= 1;
	aLMP_PTM[21].iPumpGrp	:= 2;
	aLMP_PTM[21].xActive	:= 1;
	aLMP_PTM[30].iPumpGrp	:= 3;
	aLMP_PTM[30].xActive	:= 1;
	aLMP_PTM[31].iPumpGrp	:= 3;
	aLMP_PTM[31].xActive	:= 1;
	aLMP_PTM[32].iPumpGrp	:= 3;
	aLMP_PTM[32].xActive	:= 1;
	aLMP_PTM[33].iPumpGrp	:= 3;
	aLMP_PTM[33].xActive	:= 1;
	aLMP_PTM[40].iPumpGrp	:= 4;
	aLMP_PTM[40].xActive	:= 1;
	aLMP_PTM[41].iPumpGrp	:= 4;
	aLMP_PTM[41].xActive	:= 1;
	LMP_PTM44.xActive 	:= 1;
	LMP_PTM44.iPumpGrp	:= 4;


END_IF

END_PROGRAM

// ---- POUs/p_ModbusMapRx.TcPOU
PROGRAM p_ModbusMapRx
VAR

END_VAR

(* Modbus map Rx *)
(* This goes on the PLC *)

(* To prevent misalignment when changing the modbus map, the LOTO bit should be set true
to prevent EPICS from changing these bits in the PLC *)

xLOTO := mb_Output_Coils[0];
LMP_Sys00.xOverrideMode := mb_Output_Coils[1];

//Removed pnCCD encoders from LOTO
LMP_ENC01.xENC_PWR_SW:=mb_Output_Coils[200];
LMP_ENC02.xENC_PWR_SW:=mb_Output_Coils[201];
LMP_ENC03.xENC_PWR_SW:=mb_Output_Coils[202];

IF xLOTO THEN

(* Binary controls from PLC TO EPICS *)

mb_Output_Coils[100]:=aLMP_PTM[10].i_xRunSW;
mb_Output_Coils[101]:=aLMP_PTM[11].i_xRunSW;
mb_Output_Coils[102]:=aLMP_PTM[30].i_xRunSW;
mb_Output_Coils[103]:=aLMP_PTM[31].i_xRunSW;
mb_Output_Coils[104]:=aLMP_PTM[32].i_xRunSW;
mb_Output_Coils[105]:=aLMP_PTM[33].i_xRunSW;
mb_Output_Coils[106]:=aLMP_PTM[40].i_xRunSW;
mb_Output_Coils[107]:=LMP_PTM44.i_xRunSW;
mb_Output_Coils[108]:=aLMP_PTM[41].i_xRunSW;
mb_Output_Coils[109]:=aLMP_PTM[20].i_xRunSW;
mb_Output_Coils[110]:=aLMP_PTM[21].i_xRunSW;
mb_Output_Coils[150]:=LMP_VG[10].xHV_SW;
mb_Output_Coils[151]:=LMP_VG[12].xHV_SW;
mb_Output_Coils[152]:=LMP_VG[22].xHV_SW;
mb_Output_Coils[153]:=LMP_VG[31].xHV_SW;
mb_Output_Coils[154]:=LMP_VG[13].xHV_SW;
mb_Output_Coils[155]:=LMP_VG[11].xHV_SW;
mb_Output_Coils[156]:=LMP_VG[20].xHV_SW;
mb_Output_Coils[157]:=LMP_VG[30].xHV_SW;
mb_Output_Coils[158]:=LMP_VG[43].xHV_SW;
mb_Output_Coils[159]:=LMP_VG[42].xHV_SW;
mb_Output_Coils[160]:=LMP_VG[01].xHV_SW;
mb_Output_Coils[161]:=LMP_VG[02].xHV_SW;
mb_Output_Coils[162]:=LMP_VG[41].xHV_SW;
mb_Output_Coils[163]:=LMP_VG[40].xHV_SW;
mb_Output_Coils[164]:=LMP_VG[21].xHV_SW;
mb_Output_Coils[165]:=LMP_VG[03].xHV_SW;
mb_Output_Coils[166]:=LMP_VG[04].xHV_SW;
mb_Output_Coils[167]:=LMP_VG[05].xHV_SW;

mb_Output_Coils[10]:=LMP_VGC30.xOPN_SW;
mb_Output_Coils[11]:=LMP_VGC10.xOPN_SW;
mb_Output_Coils[12]:=LMP_VRC04.xOPN_SW;
mb_Output_Coils[13]:=LMP_VRC03.xOPN_SW;
mb_Output_Coils[14]:=LMP_VRC01.xOPN_SW;
mb_Output_Coils[15]:=LMP_VRC02.xOPN_SW;
mb_Output_Coils[16]:=LMP_VRC05.xOPN_SW;
mb_Output_Coils[17]:=LMP_VRC06.xOPN_SW;
mb_Output_Coils[18]:=LMP_VRC07.xOPN_SW;
mb_Output_Coils[60]:=LMP_VCCUSR.xOPN_SW;

mb_Output_Coils[50]:=LMP_VRC01.xOvrdOpn;
mb_Output_Coils[51]:=LMP_VRC02.xOvrdOpn;
mb_Output_Coils[52]:=LMP_VRC03.xOvrdOpn;
//mb_Output_Coils[53]:=LMP_VRC04.xOvrdOpn;
mb_Output_Coils[54]:=LMP_VRC05.xOvrdOpn;
mb_Output_Coils[55]:=LMP_VRC06.xOvrdOpn;
mb_Output_Coils[56]:=LMP_VRC07.xOvrdOpn;



(* Real controls from PLC back to EPICS (32-bit) *)

MEMCPY(destAddr:=ADR(mb_PLC_Memory[100]), srcAddr:=ADR(LMP_VG[10].rVAC_SP), n:=SIZEOF(LMP_VG[10].rVAC_SP));
MEMCPY(destAddr:=ADR(mb_PLC_Memory[102]), srcAddr:=ADR(LMP_VG[12].rVAC_SP), n:=SIZEOF(LMP_VG[12].rVAC_SP));
MEMCPY(destAddr:=ADR(mb_PLC_Memory[104]), srcAddr:=ADR(LMP_VG[22].rVAC_SP), n:=SIZEOF(LMP_VG[22].rVAC_SP));
MEMCPY(destAddr:=ADR(mb_PLC_Memory[106]), srcAddr:=ADR(LMP_VG[31].rVAC_SP), n:=SIZEOF(LMP_VG[31].rVAC_SP));
MEMCPY(destAddr:=ADR(mb_PLC_Memory[108]), srcAddr:=ADR(LMP_VG[13].rVAC_SP), n:=SIZEOF(LMP_VG[13].rVAC_SP));
MEMCPY(destAddr:=ADR(mb_PLC_Memory[110]), srcAddr:=ADR(LMP_VG[11].rVAC_SP), n:=SIZEOF(LMP_VG[11].rVAC_SP));
MEMCPY(destAddr:=ADR(mb_PLC_Memory[112]), srcAddr:=ADR(LMP_VG[20].rVAC_SP), n:=SIZEOF(LMP_VG[20].rVAC_SP));
MEMCPY(destAddr:=ADR(mb_PLC_Memory[114]), srcAddr:=ADR(LMP_VG[30].rVAC_SP), n:=SIZEOF(LMP_VG[30].rVAC_SP));
MEMCPY(destAddr:=ADR(mb_PLC_Memory[116]), srcAddr:=ADR(LMP_VG[43].rVAC_SP), n:=SIZEOF(LMP_VG[43].rVAC_SP));
MEMCPY(destAddr:=ADR(mb_PLC_Memory[118]), srcAddr:=ADR(LMP_VG[42].rVAC_SP), n:=SIZEOF(LMP_VG[42].rVAC_SP));
MEMCPY(destAddr:=ADR(mb_PLC_Memory[120]), srcAddr:=ADR(LMP_VG[01].rVAC_SP), n:=SIZEOF(LMP_VG[01].rVAC_SP));
MEMCPY(destAddr:=ADR(mb_PLC_Memory[122]), srcAddr:=ADR(LMP_VG[02].rVAC_SP), n:=SIZEOF(LMP_VG[02].rVAC_SP));
MEMCPY(destAddr:=ADR(mb_PLC_Memory[124]), srcAddr:=ADR(LMP_VG[41].rVAC_SP), n:=SIZEOF(LMP_VG[41].rVAC_SP));
MEMCPY(destAddr:=ADR(mb_PLC_Memory[126]), srcAddr:=ADR(LMP_VG[40].rVAC_SP), n:=SIZEOF(LMP_VG[40].rVAC_SP));
MEMCPY(destAddr:=ADR(mb_PLC_Memory[128]), srcAddr:=ADR(LMP_VG[21].rVAC_SP), n:=SIZEOF(LMP_VG[21].rVAC_SP));
MEMCPY(destAddr:=ADR(mb_PLC_Memory[130]), srcAddr:=ADR(LMP_VG[03].rVAC_SP), n:=SIZEOF(LMP_VG[03].rVAC_SP));
MEMCPY(destAddr:=ADR(mb_PLC_Memory[132]), srcAddr:=ADR(LMP_VG[04].rVAC_SP), n:=SIZEOF(LMP_VG[04].rVAC_SP));
MEMCPY(destAddr:=ADR(mb_PLC_Memory[134]), srcAddr:=ADR(LMP_VG[05].rVAC_SP), n:=SIZEOF(LMP_VG[05].rVAC_SP));
MEMCPY(destAddr:=ADR(mb_PLC_Memory[136]), srcAddr:=ADR(LMP_VG[06].rVAC_SP), n:=SIZEOF(LMP_VG[06].rVAC_SP));
MEMCPY(destAddr:=ADR(mb_PLC_Memory[138]), srcAddr:=ADR(LMP_VG[07].rVAC_SP), n:=SIZEOF(LMP_VG[07].rVAC_SP));
MEMCPY(destAddr:=ADR(mb_PLC_Memory[140]), srcAddr:=ADR(g_rExtIlkPres), n:=SIZEOF(g_rExtIlkPres));
MEMCPY(destAddr:=ADR(mb_PLC_Memory[142]), srcAddr:=ADR(LMP_VG[32].rVAC_SP), n:=SIZEOF(LMP_VG[32].rVAC_SP));

(* Int controls to EPICS *)
(* Integer controls from PLC TO EPICS *)

mb_Output_Registers[0]:=INT_TO_WORD(LMP_VG[10].iTYPE);
mb_Output_Registers[1]:=LMP_VG[10].wPG;
mb_Output_Registers[2]:=LMP_VG[10].wHV_RO;
mb_Output_Registers[3]:=INT_TO_WORD(LMP_VG[12].iTYPE);
mb_Output_Registers[4]:=LMP_VG[12].wPG;
mb_Output_Registers[5]:=LMP_VG[12].wHV_RO;
mb_Output_Registers[6]:=INT_TO_WORD(LMP_VG[22].iTYPE);
mb_Output_Registers[7]:=LMP_VG[22].wPG;
mb_Output_Registers[8]:=LMP_VG[22].wHV_RO;
mb_Output_Registers[9]:=INT_TO_WORD(LMP_VG[31].iTYPE);
mb_Output_Registers[10]:=LMP_VG[31].wPG;
mb_Output_Registers[11]:=LMP_VG[31].wHV_RO;
mb_Output_Registers[12]:=INT_TO_WORD(LMP_VG[13].iTYPE);
mb_Output_Registers[13]:=LMP_VG[13].wPG;
mb_Output_Registers[14]:=LMP_VG[13].wHV_RO;
mb_Output_Registers[15]:=INT_TO_WORD(LMP_VG[11].iTYPE);
mb_Output_Registers[16]:=LMP_VG[11].wPG;
mb_Output_Registers[17]:=LMP_VG[11].wHV_RO;
mb_Output_Registers[18]:=INT_TO_WORD(LMP_VG[20].iTYPE);
mb_Output_Registers[19]:=LMP_VG[20].wPG;
mb_Output_Registers[20]:=LMP_VG[20].wHV_RO;
mb_Output_Registers[21]:=INT_TO_WORD(LMP_VG[30].iTYPE);
mb_Output_Registers[22]:=LMP_VG[30].wPG;
mb_Output_Registers[23]:=LMP_VG[30].wHV_RO;
mb_Output_Registers[24]:=INT_TO_WORD(LMP_VG[43].iTYPE);
mb_Output_Registers[25]:=LMP_VG[43].wPG;
mb_Output_Registers[26]:=LMP_VG[43].wHV_RO;
mb_Output_Registers[27]:=INT_TO_WORD(LMP_VG[42].iTYPE);
mb_Output_Registers[28]:=LMP_VG[42].wPG;
mb_Output_Registers[29]:=LMP_VG[42].wHV_RO;
mb_Output_Registers[30]:=INT_TO_WORD(LMP_VG[01].iTYPE);
mb_Output_Registers[31]:=LMP_VG[01].wPG;
mb_Output_Registers[32]:=LMP_VG[01].wHV_RO;
mb_Output_Registers[33]:=INT_TO_WORD(LMP_VG[02].iTYPE);
mb_Output_Registers[34]:=LMP_VG[02].wPG;
mb_Output_Registers[35]:=LMP_VG[02].wHV_RO;
mb_Output_Registers[36]:=INT_TO_WORD(LMP_VG[41].iTYPE);
mb_Output_Registers[37]:=LMP_VG[41].wPG;
mb_Output_Registers[38]:=LMP_VG[41].wHV_RO;
mb_Output_Registers[39]:=INT_TO_WORD(LMP_VG[40].iTYPE);
mb_Output_Registers[40]:=LMP_VG[40].wPG;
mb_Output_Registers[41]:=LMP_VG[40].wHV_RO;
mb_Output_Registers[42]:=INT_TO_WORD(LMP_VG[21].iTYPE);
mb_Output_Registers[43]:=LMP_VG[21].wPG;
mb_Output_Registers[44]:=LMP_VG[21].wHV_RO;
mb_Output_Registers[45]:=INT_TO_WORD(LMP_VG[03].iTYPE);
mb_Output_Registers[46]:=LMP_VG[03].wPG;
mb_Output_Registers[47]:=LMP_VG[03].wHV_RO;
mb_Output_Registers[48]:=INT_TO_WORD(LMP_VG[04].iTYPE);
mb_Output_Registers[49]:=LMP_VG[04].wPG;
mb_Output_Registers[50]:=LMP_VG[04].wHV_RO;
mb_Output_Registers[51]:=INT_TO_WORD(LMP_VG[05].iTYPE);
mb_Output_Registers[52]:=LMP_VG[05].wPG;
mb_Output_Registers[53]:=LMP_VG[05].wHV_RO;
mb_Output_Registers[54]:=INT_TO_WORD(LMP_VG[06].iTYPE);
mb_Output_Registers[55]:=LMP_VG[06].wPG;
mb_Output_Registers[56]:=LMP_VG[06].wHV_RO;
mb_Output_Registers[57]:=INT_TO_WORD(LMP_VG[07].iTYPE);
mb_Output_Registers[58]:=LMP_VG[07].wPG;
mb_Output_Registers[59]:=LMP_VG[07].wHV_RO;
mb_Output_Registers[60]:=INT_TO_WORD(g_iExtIlkGauge);
mb_Output_Registers[61]:=INT_TO_WORD(aLMP_PTM[10].i_iErrorCode);
mb_Output_Registers[62]:=INT_TO_WORD(aLMP_PTM[10].i_iWarningCode);
mb_Output_Registers[63]:=INT_TO_WORD(aLMP_PTM[11].i_iErrorCode);
mb_Output_Registers[64]:=INT_TO_WORD(aLMP_PTM[11].i_iWarningCode);
mb_Output_Registers[65]:=INT_TO_WORD(aLMP_PTM[30].i_iErrorCode);
mb_Output_Registers[66]:=INT_TO_WORD(aLMP_PTM[30].i_iWarningCode);
mb_Output_Registers[67]:=INT_TO_WORD(aLMP_PTM[31].i_iErrorCode);
mb_Output_Registers[68]:=INT_TO_WORD(aLMP_PTM[31].i_iWarningCode);
mb_Output_Registers[69]:=INT_TO_WORD(aLMP_PTM[32].i_iErrorCode);
mb_Output_Registers[70]:=INT_TO_WORD(aLMP_PTM[32].i_iWarningCode);
mb_Output_Registers[71]:=INT_TO_WORD(aLMP_PTM[33].i_iErrorCode);
mb_Output_Registers[72]:=INT_TO_WORD(aLMP_PTM[33].i_iWarningCode);
mb_Output_Registers[73]:=INT_TO_WORD(aLMP_PTM[20].i_iErrorCode);
mb_Output_Registers[74]:=INT_TO_WORD(aLMP_PTM[20].i_iWarningCode);
mb_Output_Registers[75]:=INT_TO_WORD(aLMP_PTM[21].i_iErrorCode);
mb_Output_Registers[76]:=INT_TO_WORD(aLMP_PTM[21].i_iWarningCode);
mb_Output_Registers[77]:=INT_TO_WORD(LMP_VG[32].iTYPE);
mb_Output_Registers[78]:=LMP_VG[32].wPG;
mb_Output_Registers[79]:=LMP_VG[32].wHV_RO;

ELSE

(* Binary controls from EPICS to PLC *)

aLMP_PTM[10].i_xRunSW:=mb_Output_Coils[100];
aLMP_PTM[11].i_xRunSW:=mb_Output_Coils[101];
aLMP_PTM[30].i_xRunSW:=mb_Output_Coils[102];
aLMP_PTM[31].i_xRunSW:=mb_Output_Coils[103];
aLMP_PTM[32].i_xRunSW:=mb_Output_Coils[104];
aLMP_PTM[33].i_xRunSW:=mb_Output_Coils[105];
aLMP_PTM[40].i_xRunSW:=mb_Output_Coils[106];
LMP_PTM44.i_xRunSW:=mb_Output_Coils[107];
aLMP_PTM[41].i_xRunSW:=mb_Output_Coils[108];
aLMP_PTM[20].i_xRunSW:=mb_Output_Coils[109];
aLMP_PTM[21].i_xRunSW:=mb_Output_Coils[110];
LMP_VG[10].xHV_SW:=mb_Output_Coils[150];
LMP_VG[12].xHV_SW:=mb_Output_Coils[151];
LMP_VG[22].xHV_SW:=mb_Output_Coils[152];
LMP_VG[31].xHV_SW:=mb_Output_Coils[153];
LMP_VG[13].xHV_SW:=mb_Output_Coils[154];
LMP_VG[11].xHV_SW:=mb_Output_Coils[155];
LMP_VG[20].xHV_SW:=mb_Output_Coils[156];
LMP_VG[30].xHV_SW:=mb_Output_Coils[157];
LMP_VG[43].xHV_SW:=mb_Output_Coils[158];
LMP_VG[42].xHV_SW:=mb_Output_Coils[159];
LMP_VG[01].xHV_SW:=mb_Output_Coils[160];
LMP_VG[02].xHV_SW:=mb_Output_Coils[161];
LMP_VG[41].xHV_SW:=mb_Output_Coils[162];
LMP_VG[40].xHV_SW:=mb_Output_Coils[163];
LMP_VG[21].xHV_SW:=mb_Output_Coils[164];
LMP_VG[03].xHV_SW:=mb_Output_Coils[165];
LMP_VG[04].xHV_SW:=mb_Output_Coils[166];
LMP_VG[05].xHV_SW:=mb_Output_Coils[167];

LMP_VGC30.xOPN_SW:=mb_Output_Coils[10];
LMP_VGC10.xOPN_SW:=mb_Output_Coils[11];
LMP_VRC04.xOPN_SW:=mb_Output_Coils[12];
LMP_VRC03.xOPN_SW:=mb_Output_Coils[13];
LMP_VRC01.xOPN_SW:=mb_Output_Coils[14];
LMP_VRC02.xOPN_SW:=mb_Output_Coils[15];
LMP_VRC05.xOPN_SW:=mb_Output_Coils[16];
LMP_VRC06.xOPN_SW:=mb_Output_Coils[17];
LMP_VRC07.xOPN_SW:=mb_Output_Coils[18];
LMP_VCCUSR.xOPN_SW:=mb_Output_Coils[60];

LMP_VRC01.xOvrdOpn:=mb_Output_Coils[50];
LMP_VRC02.xOvrdOpn:=mb_Output_Coils[51];
LMP_VRC03.xOvrdOpn:=mb_Output_Coils[52];
//LMP_VRC04.xOvrdOpn:=mb_Output_Coils[53];
LMP_VRC05.xOvrdOpn:=mb_Output_Coils[54];
LMP_VRC06.xOvrdOpn:=mb_Output_Coils[55];
LMP_VRC07.xOvrdOpn:=mb_Output_Coils[56];

(* Integer controls from EPICS to PLC *)

LMP_VG[10].iTYPE:=WORD_TO_INT(mb_Output_Registers[0]);
LMP_VG[10].wPG:=mb_Output_Registers[1];
LMP_VG[10].wHV_RO:=mb_Output_Registers[2];
LMP_VG[12].iTYPE:=WORD_TO_INT(mb_Output_Registers[3]);
LMP_VG[12].wPG:=mb_Output_Registers[4];
LMP_VG[12].wHV_RO:=mb_Output_Registers[5];
LMP_VG[22].iTYPE:=WORD_TO_INT(mb_Output_Registers[6]);
LMP_VG[22].wPG:=mb_Output_Registers[7];
LMP_VG[22].wHV_RO:=mb_Output_Registers[8];
LMP_VG[31].iTYPE:=WORD_TO_INT(mb_Output_Registers[9]);
LMP_VG[31].wPG:=mb_Output_Registers[10];
LMP_VG[31].wHV_RO:=mb_Output_Registers[11];
LMP_VG[13].iTYPE:=WORD_TO_INT(mb_Output_Registers[12]);
LMP_VG[13].wPG:=mb_Output_Registers[13];
LMP_VG[13].wHV_RO:=mb_Output_Registers[14];
LMP_VG[11].iTYPE:=WORD_TO_INT(mb_Output_Registers[15]);
LMP_VG[11].wPG:=mb_Output_Registers[16];
LMP_VG[11].wHV_RO:=mb_Output_Registers[17];
LMP_VG[20].iTYPE:=WORD_TO_INT(mb_Output_Registers[18]);
LMP_VG[20].wPG:=mb_Output_Registers[19];
LMP_VG[20].wHV_RO:=mb_Output_Registers[20];
LMP_VG[30].iTYPE:=WORD_TO_INT(mb_Output_Registers[21]);
LMP_VG[30].wPG:=mb_Output_Registers[22];
LMP_VG[30].wHV_RO:=mb_Output_Registers[23];
LMP_VG[43].iTYPE:=WORD_TO_INT(mb_Output_Registers[24]);
LMP_VG[43].wPG:=mb_Output_Registers[25];
LMP_VG[43].wHV_RO:=mb_Output_Registers[26];
LMP_VG[42].iTYPE:=WORD_TO_INT(mb_Output_Registers[27]);
LMP_VG[42].wPG:=mb_Output_Registers[28];
LMP_VG[42].wHV_RO:=mb_Output_Registers[29];
LMP_VG[01].iTYPE:=WORD_TO_INT(mb_Output_Registers[30]);
LMP_VG[01].wPG:=mb_Output_Registers[31];
LMP_VG[01].wHV_RO:=mb_Output_Registers[32];
LMP_VG[02].iTYPE:=WORD_TO_INT(mb_Output_Registers[33]);
LMP_VG[02].wPG:=mb_Output_Registers[34];
LMP_VG[02].wHV_RO:=mb_Output_Registers[35];
LMP_VG[41].iTYPE:=WORD_TO_INT(mb_Output_Registers[36]);
LMP_VG[41].wPG:=mb_Output_Registers[37];
LMP_VG[41].wHV_RO:=mb_Output_Registers[38];
LMP_VG[40].iTYPE:=WORD_TO_INT(mb_Output_Registers[39]);
LMP_VG[40].wPG:=mb_Output_Registers[40];
LMP_VG[40].wHV_RO:=mb_Output_Registers[41];
LMP_VG[21].iTYPE:=WORD_TO_INT(mb_Output_Registers[42]);
LMP_VG[21].wPG:=mb_Output_Registers[43];
LMP_VG[21].wHV_RO:=mb_Output_Registers[44];
LMP_VG[03].iTYPE:=WORD_TO_INT(mb_Output_Registers[45]);
LMP_VG[03].wPG:=mb_Output_Registers[46];
LMP_VG[03].wHV_RO:=mb_Output_Registers[47];
LMP_VG[04].iTYPE:=WORD_TO_INT(mb_Output_Registers[48]);
LMP_VG[04].wPG:=mb_Output_Registers[49];
LMP_VG[04].wHV_RO:=mb_Output_Registers[50];
LMP_VG[05].iTYPE:=WORD_TO_INT(mb_Output_Registers[51]);
LMP_VG[05].wPG:=mb_Output_Registers[52];
LMP_VG[05].wHV_RO:=mb_Output_Registers[53];
LMP_VG[06].iTYPE:=WORD_TO_INT(mb_Output_Registers[54]);
LMP_VG[06].wPG:=mb_Output_Registers[55];
LMP_VG[06].wHV_RO:=mb_Output_Registers[56];
LMP_VG[07].iTYPE:=WORD_TO_INT(mb_Output_Registers[57]);
LMP_VG[07].wPG:=mb_Output_Registers[58];
LMP_VG[07].wHV_RO:=mb_Output_Registers[59];
g_iExtIlkGauge   :=WORD_TO_INT(mb_Output_Registers[60]);
LMP_VG[32].iTYPE:=WORD_TO_INT(mb_Output_Registers[77]);
LMP_VG[32].wPG:=mb_Output_Registers[78];
LMP_VG[32].wHV_RO:=mb_Output_Registers[79];


(* Real controls from EPICS (32-bit) to PLC *)

MEMCPY(destAddr:=ADR(LMP_VG[10].rVAC_SP), srcAddr:=ADR(mb_PLC_Memory[100]), n:=SIZEOF(LMP_VG[10].rVAC_SP));
MEMCPY(destAddr:=ADR(LMP_VG[12].rVAC_SP), srcAddr:=ADR(mb_PLC_Memory[102]), n:=SIZEOF(LMP_VG[12].rVAC_SP));
MEMCPY(destAddr:=ADR(LMP_VG[22].rVAC_SP), srcAddr:=ADR(mb_PLC_Memory[104]), n:=SIZEOF(LMP_VG[22].rVAC_SP));
MEMCPY(destAddr:=ADR(LMP_VG[31].rVAC_SP), srcAddr:=ADR(mb_PLC_Memory[106]), n:=SIZEOF(LMP_VG[31].rVAC_SP));
MEMCPY(destAddr:=ADR(LMP_VG[13].rVAC_SP), srcAddr:=ADR(mb_PLC_Memory[108]), n:=SIZEOF(LMP_VG[13].rVAC_SP));
MEMCPY(destAddr:=ADR(LMP_VG[11].rVAC_SP), srcAddr:=ADR(mb_PLC_Memory[110]), n:=SIZEOF(LMP_VG[11].rVAC_SP));
MEMCPY(destAddr:=ADR(LMP_VG[20].rVAC_SP), srcAddr:=ADR(mb_PLC_Memory[112]), n:=SIZEOF(LMP_VG[20].rVAC_SP));
MEMCPY(destAddr:=ADR(LMP_VG[30].rVAC_SP), srcAddr:=ADR(mb_PLC_Memory[114]), n:=SIZEOF(LMP_VG[30].rVAC_SP));
MEMCPY(destAddr:=ADR(LMP_VG[43].rVAC_SP), srcAddr:=ADR(mb_PLC_Memory[116]), n:=SIZEOF(LMP_VG[43].rVAC_SP));
MEMCPY(destAddr:=ADR(LMP_VG[42].rVAC_SP), srcAddr:=ADR(mb_PLC_Memory[118]), n:=SIZEOF(LMP_VG[42].rVAC_SP));
MEMCPY(destAddr:=ADR(LMP_VG[01].rVAC_SP), srcAddr:=ADR(mb_PLC_Memory[120]), n:=SIZEOF(LMP_VG[01].rVAC_SP));
MEMCPY(destAddr:=ADR(LMP_VG[02].rVAC_SP), srcAddr:=ADR(mb_PLC_Memory[122]), n:=SIZEOF(LMP_VG[02].rVAC_SP));
MEMCPY(destAddr:=ADR(LMP_VG[41].rVAC_SP), srcAddr:=ADR(mb_PLC_Memory[124]), n:=SIZEOF(LMP_VG[41].rVAC_SP));
MEMCPY(destAddr:=ADR(LMP_VG[40].rVAC_SP), srcAddr:=ADR(mb_PLC_Memory[126]), n:=SIZEOF(LMP_VG[40].rVAC_SP));
MEMCPY(destAddr:=ADR(LMP_VG[21].rVAC_SP), srcAddr:=ADR(mb_PLC_Memory[128]), n:=SIZEOF(LMP_VG[21].rVAC_SP));
MEMCPY(destAddr:=ADR(LMP_VG[03].rVAC_SP), srcAddr:=ADR(mb_PLC_Memory[130]), n:=SIZEOF(LMP_VG[03].rVAC_SP));
MEMCPY(destAddr:=ADR(LMP_VG[04].rVAC_SP), srcAddr:=ADR(mb_PLC_Memory[132]), n:=SIZEOF(LMP_VG[04].rVAC_SP));
MEMCPY(destAddr:=ADR(LMP_VG[05].rVAC_SP), srcAddr:=ADR(mb_PLC_Memory[134]), n:=SIZEOF(LMP_VG[05].rVAC_SP));
MEMCPY(destAddr:=ADR(LMP_VG[06].rVAC_SP), srcAddr:=ADR(mb_PLC_Memory[136]), n:=SIZEOF(LMP_VG[06].rVAC_SP));
MEMCPY(destAddr:=ADR(LMP_VG[07].rVAC_SP), srcAddr:=ADR(mb_PLC_Memory[138]), n:=SIZEOF(LMP_VG[07].rVAC_SP));
MEMCPY(destAddr:=ADR(g_rExtIlkPres), srcAddr:=ADR(mb_PLC_Memory[140]), n:=SIZEOF(g_rExtIlkPres));
MEMCPY(destAddr:=ADR(LMP_VG[32].rVAC_SP), srcAddr:=ADR(mb_PLC_Memory[142]), n:=SIZEOF(LMP_VG[32].rVAC_SP));
END_IF

(***********************************************************)

END_PROGRAM

// ---- POUs/p_Autosave.TcPOU
PROGRAM p_Autosave
VAR
	iIndex: INT;
END_VAR

(* If first pass, copy all persistent variables (which should be intialized to old values) back into the operational variables *)
IF LMP_SYS00.xFirstScan THEN
	FOR iIndex:=0 TO 50 DO
		LMP_VG[iIndex].iTYPE := gp_LMP_VG[iIndex].iTYPE;
		LMP_VG[iIndex].rFULL_SCALE := gp_LMP_VG[iIndex].rFULL_SCALE;
		LMP_VG[iIndex].rPRO_SP := gp_LMP_VG[iIndex].rPRO_SP;
		LMP_VG[iIndex].rVAC_SP := gp_LMP_VG[iIndex].rVAC_SP;
		LMP_VG[iIndex].wHV_RO := gp_LMP_VG[iIndex].wHV_RO;
		LMP_VG[iIndex].wPG := gp_LMP_VG[iIndex].wPG;
	END_FOR
ELSE
	FOR iIndex:=0 TO 50 DO
		gp_LMP_VG[iIndex].iTYPE			:=	LMP_VG[iIndex].iTYPE;
		gp_LMP_VG[iIndex].rFULL_SCALE	:=	LMP_VG[iIndex].rFULL_SCALE;
		gp_LMP_VG[iIndex].rPRO_SP		:=	LMP_VG[iIndex].rPRO_SP;
		gp_LMP_VG[iIndex].rVAC_SP		:=	LMP_VG[iIndex].rVAC_SP;
		gp_LMP_VG[iIndex].wHV_RO		:=	LMP_VG[iIndex].wHV_RO;
		gp_LMP_VG[iIndex].wPG			:=	LMP_VG[iIndex].wPG;
	END_FOR
END_IF

END_PROGRAM

// ---- POUs/P_Serial_PTM_IO.TcPOU
PROGRAM P_Serial_PTM_IO
VAR
	fb_IC_P1_PfeifferCom : FB_PFEIFFER_COM;
	fb_R10_A_P1_OerlikonTD20 : FB_Oerlikon_TD20_COM;

	xFirstScan: BOOL := TRUE;
END_VAR

(*
This program takes care of calling the FB_PFEIFFER_COM blocks
 which are responsible for carrying out the IO communications over serial.
 It is placed in it's own PLC task to give it independence from when the 
 supervisor programs.

This program is called from A00_MAIN
 
*)

// Calling port specific communication function blocks

// IC EP6002 - Port 1
fb_IC_P1_PfeifferCom(astPfeifferControl := g_astPfe_CTRL,
				 astPfeifferStatus	:= g_astPfe_RBK,
				 afbPfeifferSerialDriver := g_afbPfe_SerialDriver,

				SerialRXBuffer:= IC_P1_SerialRXBuffer,
				SerialTXBuffer:= IC_P1_SerialTXBuffer);

// R10 A - Port 1				
fb_R10_A_P1_OerlikonTD20(astTD20Status := g_astTD20_RBK,
				fbTD20SerialDriver := g_astTD20_SerialDriver,

				SerialRXBuffer := R10_A_P1_SerialRXBuffer,
				 SerialTXBuffer := R10_A_P1_SerialTXBuffer);

END_PROGRAM

// ---- POUs/p_SoftIOMap.TcPOU
PROGRAM p_SoftIOMap
VAR
	
	fbPfeifferToPTM : FB_PFEIFFER_TO_PTM;

	Oerlikon_to_PTM44 : FB_OERLIKON_TO_PTM;
	
	iDummy	: REAL;
	xDummy	: BOOL;
	i       : INT;

END_VAR
VAR_INPUT
END_VAR

(* Soft to Hard IO Tag Map *)
(* Hard input tags are copied to Soft inputs tags, Soft output tags are copied to *)
(* Hard input tags. Soft IO tags are used within the program and can be modified as needed. *)
(* Added to this list to include dummy variables for the IO points so they wold be mapped to the correct task *)

(* Mapping the PTM names to something more user friendly *)
(* 6002 *)
fbPfeifferToPTM(iq_stPfeiffer_ctrl:= g_astPfe_CTRL[1], iq_stPfeiffer_stat := g_astPfe_RBK[1], iq_stPTM := aLMP_PTM[10]);
fbPfeifferToPTM(iq_stPfeiffer_ctrl:= g_astPfe_CTRL[2], iq_stPfeiffer_stat := g_astPfe_RBK[2], iq_stPTM := aLMP_PTM[11]);
fbPfeifferToPTM(iq_stPfeiffer_ctrl:= g_astPfe_CTRL[3], iq_stPfeiffer_stat := g_astPfe_RBK[3], iq_stPTM := aLMP_PTM[30]);
fbPfeifferToPTM(iq_stPfeiffer_ctrl:= g_astPfe_CTRL[4], iq_stPfeiffer_stat := g_astPfe_RBK[4], iq_stPTM := aLMP_PTM[31]);
fbPfeifferToPTM(iq_stPfeiffer_ctrl:= g_astPfe_CTRL[5], iq_stPfeiffer_stat := g_astPfe_RBK[5], iq_stPTM := aLMP_PTM[32]);
fbPfeifferToPTM(iq_stPfeiffer_ctrl:= g_astPfe_CTRL[6], iq_stPfeiffer_stat := g_astPfe_RBK[6], iq_stPTM := aLMP_PTM[33]);
fbPfeifferToPTM(iq_stPfeiffer_ctrl:= g_astPfe_CTRL[7], iq_stPfeiffer_stat := g_astPfe_RBK[7], iq_stPTM := aLMP_PTM[20]);
fbPfeifferToPTM(iq_stPfeiffer_ctrl:= g_astPfe_CTRL[8], iq_stPfeiffer_stat := g_astPfe_RBK[8], iq_stPTM := aLMP_PTM[21]);
fbPfeifferToPTM(iq_stPfeiffer_ctrl:= g_astPfe_CTRL[9], iq_stPfeiffer_stat := g_astPfe_RBK[9], iq_stPTM := aLMP_PTM[40]);
fbPfeifferToPTM(iq_stPfeiffer_ctrl:= g_astPfe_CTRL[10], iq_stPfeiffer_stat := g_astPfe_RBK[10], iq_stPTM := aLMP_PTM[41]);

Oerlikon_to_PTM44(iq_stOerlikon_stat:=g_astTD20_RBK, iq_stPTM:= LMP_PTM44);

(* Controls *)
(* EP2339 *)
	DiscIO_LRS_EB3Ch01:=LMP_VRC01.xOPN_DO;
	DiscIO_LRS_EB3Ch04:=LMP_VRC02.xOPN_DO;
	DiscIO_LRS_EB3Ch07:=LMP_VRC03.xOPN_DO;
	DiscIO_LRS_EB3Ch10:=LMP_VRC04.xOPN_DO;
	DiscIO_LRS_EB3Ch13:=LMP_VRC05.xOPN_DO;
	DiscIO_LRS_EB4Ch01:=LMP_VRC06.xOPN_DO;
	DiscIO_LRS_EB4Ch04:=LMP_VRC07.xOPN_DO;
	//User valve
	DiscIO_GJ_EB3Ch04:=LMP_VCCUSR.xOPN_DO;


(* HV Enables *)
(* EP2624 *)
	RelayO_DET_EB3Ch01 := LMP_RO[30];
	RelayO_DET_EB3Ch02 := LMP_RO[31];
	RelayO_DET_EB3Ch03 := LMP_RO[32];
	RelayO_DET_EB3Ch04 := LMP_RO[33];

	RelayO_DET_EB5Ch01 := LMP_RO[34];
	RelayO_DET_EB5Ch02 := LMP_RO[35];
	RelayO_DET_EB5Ch03 := LMP_RO[36];
	RelayO_DET_EB5Ch04 := LMP_RO[37];	
	
	
	RelayO_IC_EB3Ch01 := LMP_RO[20];
	RelayO_IC_EB3Ch02 := LMP_RO[21];
	RelayO_IC_EB3Ch03 := LMP_RO[22];
	RelayO_IC_EB3Ch04 := FALSE;
		
	RelayO_GJ_EB1Ch01 := LMP_RO[40];
	RelayO_GJ_EB1Ch02 := LMP_RO[41];
	RelayO_GJ_EB1Ch03 := LMP_RO[42];
	RelayO_GJ_EB1Ch04 := LMP_RO[43];

(* Readbacks *)

(* PLC bus *)
xDummy := DI_Term4_Ch1;

(* Valves *)
(* EP2339 *)
	LMP_VGC30.i_xOpnLS:=DiscIO_DET_EB4Ch02;
	LMP_VGC30.i_xClsLS:=DiscIO_DET_EB4Ch03;

	LMP_VGC10.i_xOpnLS:=DiscIO_IC_EB4Ch14;
	LMP_VGC10.i_xClsLS:=DiscIO_IC_EB4Ch15;
	
	LMP_VRC01.i_xOpnLS:=DiscIO_LRS_EB3Ch02;
	LMP_VRC01.i_xClsLS:=DiscIO_LRS_EB3Ch03;
	
	LMP_VRC02.i_xOpnLS:=DiscIO_LRS_EB3Ch05;
	LMP_VRC02.i_xClsLS:=DiscIO_LRS_EB3Ch06;
	
	LMP_VRC03.i_xOpnLS:=DiscIO_LRS_EB3Ch08;
	LMP_VRC03.i_xClsLS:=DiscIO_LRS_EB3Ch09;
	
	LMP_VRC04.i_xOpnLS:=DiscIO_LRS_EB3Ch11;
	LMP_VRC04.i_xClsLS:=DiscIO_LRS_EB3Ch12;
	
	LMP_VRC05.i_xOpnLS:=DiscIO_LRS_EB3Ch14;
	LMP_VRC05.i_xClsLS:=DiscIO_LRS_EB3Ch15;
	
	LMP_VRC06.i_xOpnLS:=DiscIO_LRS_EB4Ch02;
	LMP_VRC06.i_xClsLS:=DiscIO_LRS_EB4Ch03;
	
	LMP_VRC07.i_xOpnLS:=DiscIO_LRS_EB4Ch05;
	LMP_VRC07.i_xClsLS:=DiscIO_LRS_EB4Ch06;
	
	
(*	H2E_VGC01.i_xOpnLS:=DiscIO_DET_EB1Ch05;
	H2E_VGC01.i_xClsLS:=DiscIO_DET_EB1Ch06;
	
	H2E_VGC02.i_xOpnLS:=DiscIO_H2E_EB1Ch02;
	H2E_VGC02.i_xClsLS:=DiscIO_H2E_EB1Ch03; *)

	
(* Gauges *)

(* Interaction Chamber *)
(* EP3174 *)
	LMP_VG[20].iPRESS_R := AI_IC_EB2Ch01;
	LMP_VG[21].iPRESS_R := AI_IC_EB2Ch02;
	LMP_VG[22].iPRESS_R := AI_IC_EB2Ch03;
	LMP_VG[23].iPRESS_R := AI_IC_EB2Ch04;
(* Roughing lines *)
(* EP3174 *)
	LMP_VG[01].iPRESS_R := AI_LRS_EB1Ch01;
	LMP_VG[02].iPRESS_R := AI_LRS_EB1Ch02;
	LMP_VG[03].iPRESS_R := AI_LRS_EB1Ch03;
	LMP_VG[04].iPRESS_R := AI_LRS_EB1Ch04;
	LMP_VG[05].iPRESS_R := AI_LRS_EB2Ch01;
	LMP_VG[06].iPRESS_R := AI_LRS_EB2Ch02;
	LMP_VG[07].iPRESS_R := AI_LRS_EB2Ch03;
	LMP_VG[08].iPRESS_R := AI_LRS_EB2Ch04;


(* Detector chamber *)
(* EP3174 *)
	LMP_VG[30].iPRESS_R := AI_DET_EB2Ch01;
	LMP_VG[31].iPRESS_R := AI_DET_EB2Ch02;
	LMP_VG[32].iPRESS_R := AI_DET_EB2Ch03;
	LMP_VG[33].iPRESS_R := AI_DET_EB2Ch04;

(* Gas Jet *)
(* EP3174 *)
	LMP_VG[40].iPRESS_R := AI_GJ_EB2Ch01;
	LMP_VG[41].iPRESS_R := AI_GJ_EB2Ch02;
	LMP_VG[42].iPRESS_R := AI_GJ_EB2Ch03;
	LMP_VG[43].iPRESS_R := AI_GJ_EB2Ch04;

(* H2E *)
//	H2E_VG01.iPRESS_R := AI_H2E_EB2Ch01; 
//	H2E_VG02.iPRESS_R := AI_H2E_EB2Ch02;

(* Encoders & SXD PS permissive *)
(* EP2624 *)
RelayO_DET_EB5Ch01 := LMP_ENC01.xENC_PWR;
RelayO_DET_EB5Ch02 := LMP_ENC02.xENC_PWR;
RelayO_DET_EB5Ch03 := LMP_ENC03.xENC_PWR;
RelayO_DET_EB5Ch04 := g_xExtIlkRO;

(* EtherCAT Slave interface *)
(* MPS Outputs to Main PLC *)
LAMP_MPS_1 := LMP_VGC10.i_xOpnLS;
LAMP_MPS_2 := LMP_VGC30.i_xOpnLS;
LAMP_MPS_3 := LMP_VGC30.i_xClsLS;
LAMP_MPS_4 := H2E_VGC01.i_xOpnLS AND H2E_VGC02.i_xOpnLS ;
LAMP_MPS_5 := FALSE;
LAMP_MPS_6 := FALSE;
LAMP_MPS_7 := FALSE;
LAMP_MPS_8 := FALSE;


(* LAMP Up/Downstream Vars *)
LAMP_BCO_1 := LMP_VG[50].xPRESS_OK; // Pressure valid boolean
LAMP_BCO_2 := LMP_VG[21].xPRESS_OK; // Pressure valid boolean
LAMP_BCO_3 := LMP_VG[21].xAT_VAC;
LAMP_BCO_4 := FALSE;
LAMP_BCO_5 := FALSE;
LAMP_BCO_6 := FALSE;
LAMP_BCO_7 := FALSE;
LAMP_BCO_8 := FALSE;

xDummy := LAMP_BRB_1; 
xDummy := LAMP_BRB_2;
xDummy := LAMP_BRB_3;
xDummy := LAMP_BRB_4;
xDummy := LAMP_BRB_5;
xDummy := LAMP_BRB_6;
xDummy := LAMP_BRB_7;
xDummy := LAMP_BRB_8;

q_rLampAuxVG1 	:= LMP_VG[50].rPRESS;
q_rLampAuxVG2	:= LMP_VG[21].rPRESS;
q_rLampAuxVG3	:= LMP_VG[10].rPRESS;
q_rLampAuxVG4	:= LMP_VG[10].rPRESS;

iDummy := i_rAuxVG1;
iDummy := i_rAuxVG2;
iDummy := i_rAuxVG3;
iDummy := i_rAuxVG4;

END_PROGRAM

// ---- POUs/p_PTMSup.TcPOU
PROGRAM p_PTMSup
VAR
	xRESET          :   BOOL := FALSE;
	fb_LMP_PTM		:	FB_PFEIFFER_PTM;

	DP_PTM_ILK : TOF;
	IC_PTM_ILK : TOF;
	DET_PTM_ILK : TOF;
END_VAR

//Simplified interlocks to *only* be based on foreline press - 6/2016

(* DP Pump Interlocks *)
DP_PTM_ILK.PT := T#15S;
DP_PTM_ILK.IN := LMP_VG[6].xAT_VAC;
DP_PTM_ILK();
aLMP_PTM[10].xExtRunOk := DP_PTM_ILK.Q;
aLMP_PTM[11].xExtRunOk := aLMP_PTM[10].xExtRunOk;

(* IC Pump interlocks *)
IC_PTM_ILK.PT := T#15s;
IC_PTM_ILK.IN := LMP_VG[6].xAT_VAC OR LMP_VG[3].xAT_VAC;
IC_PTM_ILK();

aLMP_PTM[40].xExtRunOk := IC_PTM_ILK.Q;
aLMP_PTM[41].xExtRunOk := aLMP_PTM[40].xExtRunOk;
aLMP_PTM[20].xExtRunOk := aLMP_PTM[40].xExtRunOk;
aLMP_PTM[21].xExtRunOk := aLMP_PTM[40].xExtRunOk;

(* Detector Pumps *)
DET_PTM_ILK.PT := T#15s;
DET_PTM_ILK.IN := LMP_VG[5].xAT_VAC;
DET_PTM_ILK();

aLMP_PTM[30].xExtRunOk	:=	DET_PTM_ILK.Q;
aLMP_PTM[31].xExtRunOk	:=	aLMP_PTM[30].xExtRunOk;
aLMP_PTM[32].xExtRunOk	:=	aLMP_PTM[30].xExtRunOk;
aLMP_PTM[33].xExtRunOk	:=	aLMP_PTM[30].xExtRunOk;

(* Control function blocks *)
(*Differential pumping section *)
fb_LMP_PTM(iq_stPTM:= aLMP_PTM[10]);
fb_LMP_PTM(iq_stPTM:= aLMP_PTM[11]);

(* Interaction Chamber *)
fb_LMP_PTM(iq_stPTM:= aLMP_PTM[20]);
fb_LMP_PTM(iq_stPTM:= aLMP_PTM[21]);

(* Detector Chamber *)
fb_LMP_PTM(iq_stPTM:= aLMP_PTM[30]);
fb_LMP_PTM(iq_stPTM:= aLMP_PTM[31]);
fb_LMP_PTM(iq_stPTM:= aLMP_PTM[32]);
fb_LMP_PTM(iq_stPTM:= aLMP_PTM[33]);
(* pnCCD Chamber *)

(* Gas Jet *)
fb_LMP_PTM(iq_stPTM:= aLMP_PTM[40]);
fb_LMP_PTM(iq_stPTM:= aLMP_PTM[41]);

END_PROGRAM

// ---- POUs/p_GaugeSup.TcPOU
PROGRAM p_GaugeSup
VAR
(* Change the gauge types here, and that's all you have to do! *)

	i	:	INT := 0;

	LMP_GPI00	:	ST_VG; (* simulation pirani *)


	fb_LMP_GPI_D1 : FB_Dumb_Gauge;

	fb_LMP_VG : ARRAY[1..50] OF FB_GGO;
	
    fb_H2E_VG : FB_903;

	catch: INT;
    H2E_GPI00: ST_VG;

END_VAR

(* Dummy pirani setup *)
LMP_GPI00.xPRESS_OK := TRUE;

fb_LMP_GPI_D1(iq_stPG:=LMP_GPI_D1, i_stPGA:= LMP_VG[20], i_stPGB:=LMP_VG[01], i_stVRCA:=LMP_VRC05, i_stVRCB:=LMP_VRC02);

(* Control function blocks *)

LMP_VG[50].rPRESS := 1E-3;
LMP_VG[50].iTYPE := 4;
LMP_VG[50].xPRESS_OK := TRUE;

FOR i:=1 TO 50 DO
fb_LMP_VG[i](i_iIndex:=i, iq_astGauges := LMP_VG, iq_axHV_RO:=LMP_RO);
END_FOR;
IF i >50 THEN i:=1; catch := catch +1; END_IF

H2E_GPI00.rPRESS := 1E-3;
H2E_GPI00.xPRESS_OK := TRUE;

//fb_H2E_VG(IG:=H2E_VG01,PG:=H2E_GPI00);
//fb_H2E_VG(IG:=H2E_VG02,PG:=H2E_GPI00);

END_PROGRAM

// ---- POUs/p_ValveSup.TcPOU
PROGRAM p_ValveSup
VAR
	fbLMP_VRC01	:	FB_VRC_LAMP;
	fbLMP_VRC02	:	FB_VRC_LAMP;
	fbLMP_VRC03	:	FB_VRC_LAMP;
	fbLMP_VRC04	:	FB_VRC_OK_CLS;
	fbLMP_VRC05	:	FB_VRC_LAMP;
	fbLMP_VRC06	:	FB_VRC_LAMP;
	fbLMP_VRC07	:	FB_VRC_LAMP;
	fbLMP_VRC08	:	FB_VRC_LAMP;

	fbLMP_VGC30 :   FB_VGC;
	
	fbLMP_VCCUSR :  FB_VCC;

END_VAR

(* Interlock declarations *)

g_stSystem:= LMP_Sys00;

(* User valve *)
LMP_VCCUSR.xOPN_OK := TRUE;

LMP_VRC02.xOPN_OK := F_VRC_DIODE_ILK(i_stPGA:=LMP_VG[3], i_stPGB:=LMP_VG[1]);
LMP_VRC01.xOPN_OK := LMP_VRC02.i_xOpnLS AND F_VRC_DIODE_ILK(i_stPGA:=LMP_VG[3], i_stPGB:=LMP_VG[1]);


(* Interlock for VRC 06: If DET, IC and foreline piranis > 0.1 torr, DET and IC pressures must be within 
 one order of magnitude *)

(* May implement logic here at some point? *)
LMP_VRC05.xOPN_OK := TRUE;

LMP_VRC06.xOPN_OK := ( LMP_VG[20].rPRESS < 0.1 AND LMP_VG[3].rPRESS < 0.1 )
	OR F_VALVE_REL_ILK(i_stUSG:=LMP_VG[3], i_stDSG:=LMP_VG[5], i_iOrdersMagnitude:=1);
							
LMP_VRC07.xOPN_OK := LMP_VG[2].rPRESS < 0.5;

LMP_VRC03.xOPN_OK := F_VRC_DIODE_ILK (i_stPGA:=LMP_VG[4], i_stPGB:=LMP_VG[2]); //AND LMP_VRC04.i_xOpnLS (*commented b/c VRC04 has no readback*)

